(* CODESYS project BATW_Base0.0.0.33.library
   Company: Beckhoff Automation
   DefaultNamespace: BATW_Base
   Version: 0.0.0.33
   Placeholder: BATW_Base
   Author: BATW
   Description: Base library of BATW use
   Title: BATW_Base

Project tree, tasks and I/O mapping:
  libraries: Common Behaviour Model, * (3S - Smart Software Solutions GmbH); Tc2_Standard, * (Beckhoff Automation GmbH); Tc2_System, * (Beckhoff Automation GmbH); Tc2_Utilities, * (Beckhoff Automation GmbH); Tc3_EventLogger, * (Beckhoff Automation GmbH); Tc3_JsonXml, * (Beckhoff Automation GmbH); Tc3_Module, * (Beckhoff Automation GmbH)
  CBML_BASE/
    Behaviour-Model_Enums_STATE.png
    function block FB_ActionBasic [ST]: ControlCleanupAction, ControlCyclicAction, ControlExitAction, ControlResetAction, ControlStartAction, CleanupAction, CyclicAction, ExitAction, ResetAction, StartAction, IBehaviourModel, Get_ModelState, GetName
    function block FB_ActionBasic_Logger [ST]: M_ClearAlarm, M_ConfirmAlarm, M_ConnectAlarmLogger, M_RaiseAlarm, M_SetAlarmEvent, pAlarmState, M_AddEventMsg, M_ConnectMsgLogger, M_SetMessageEvent, M_AddJsonMsg, M_ConnectJsonMsgLogger
    interface I_BaseElement: Get_ModelState, GetName, IBehaviourModel
  00000000-0000-0000-0000-000000000000|CBML_BASE\Behaviour-Model_Enums_STATE.png
  Componets/
    DUTs/
      data type E_CylinderType
      data type ST_CylinderPara
    DUTs_Motor/
      data type ST_MotorPara
    function block FB_Cylinder [ST]: CleanupAction, CyclicAction, ExitAction, ResetAction, StartAction, EnableSimulation, IsDoubleValve, M_Extend, M_GetErrorMsg, M_Reset, M_Retract
    function block FB_Motor [ST]: CleanupAction, CyclicAction, ExitAction, ResetAction, StartAction, M_MotorStop, M_MoveBackward, M_MoveForward, M_Reset
  EventLogger/
    _Interface/
      Exporter/
        interface ITF_EventLogger_Exporter: M_ExportCSV
        interface ITF_EventLogger_Exporter_Carrier: M_ConnectExporter
      Logger/
        interface ITF_EventLogger_Alarm: M_ClearAlarm, M_ConfirmAlarm, M_RaiseAlarm, M_SetAlarmEvent, pAlarmState
        interface ITF_EventLogger_Alarm_Carrier: M_ClearAlarm, M_ConfirmAlarm, M_ConnectAlarmLogger, M_RaiseAlarm, M_SetAlarmEvent, pAlarmState
        interface ITF_EventLogger_Message: M_AddEventMsg, M_SetMessageEvent
        interface ITF_EventLogger_Message_Carrier: M_AddEventMsg, M_ConnectMsgLogger, M_SetMessageEvent
    _Test/
      program Demo_EventLogger [ST]
      function block FB_LoggerTest [ST]
    DUTs/
      data type E_EventExportType
      data type E_EventLanguage
      data type ST_AlarmEvent_State
    global variables EventLogger_Parameter
    function block FB_EventLogger_Alarm [ST]: M_ClearAlarm, M_ConfirmAlarm, M_RaiseAlarm, M_SetAlarmEvent, pAlarmState
    function block FB_EventLogger_Exporter [ST]: CleanupAction, CyclicAction, StartAction, M_SetCSV, M_SetExportLanguage, M_SetExportParameter
    function block FB_EventLogger_Message [ST]: M_AddEventMsg, M_SetMessageEvent
    program PRG_EventLogger [ST]: M_ExportLoggedEvent_Off, M_ExportLoggedEvent_On, M_ExportLoggedEvent_State, M_AlarmEvent_Init, M_MessageEvent_Init
  IO-Module/
    EL1889/
      data type ST_EL1889
      data type ST_EL1889_InfoData
      data type ST_EL1889_WcState
    EL2889/
      data type ST_EL2889
  JsonMsgLogger/
    _Interface/
      Client/
        interface ITF_AddJsonMsg_Behavior: M_AddJsonMsg
        interface ITF_GetJsonMsg_Behavior: M_GetJsonMsg
        interface ITF_JsonMSg_Carrier: M_ConnectJsonMsgLogger
        interface ITF_JsonMsg_Logger: M_AddJsonMsg, M_GetJsonMsg, pQueueAmount
      Server/
        interface ITF_JsonMsg_Handler: M_AttachJsonMsgLogger
    _Test/
      program Demo_JsonMsg [ST]
      function block FB_UserUnit [ST]
    Basic_Json/
      function block FB_Json_Converter [ST]: JsonStrToObj, ObjToJsonStr
      data type ST_Json_MsgLogger
    Basic_Queue/
      function block FB_Queue [ST]: dequeueElement, enqueueElement, enqueueElementfromHead, readElementbyIndex, readNextElement, releaseQueue, changeCurrentbyIndex, checkInputErr, deleteElement, moveCurrent2Next, moveCurrent2Prev, bIsQueueCreated, getDataTypebyIndex, getNextDataType, pGetHead, pGetTail, udiGetQueuedAmount
      data type ST_Queue
    data type E_HandlerQueueType
    data type E_LoggerQueueType
    data type E_OS_Type
    function block FB_JsonMsg_Handler [ST]: CleanupAction, CyclicAction, StartAction, M_AddJsonMsg, M_GetFilePathByTime, M_HandleMessage, FB_init, M_AttachJsonMsgLogger, M_SetFilePath
    function block FB_JsonMsg_Logger [ST]: M_AddJsonMsg, M_GetJsonMsg, pQueueAmount
    global variables JsonMsg_Parameter
    program PRG_JsonMsg [ST]: M_JsonMsg_Init, M_JsonMsg_SetFilePath
  POUs/
    program Demo [ST]
  Utilities/
    function block FB_EdgeDetect [ST]
  VISUs/
*)

// Componets/DUTs/E_CylinderType
{attribute 'qualified_only'}
{attribute 'strict'}
TYPE
    E_CylinderType :
    (
        Undefined    := 0,
        NoSensor     := 1,
        FrontSensor  := 2,
        RearSensor   := 3,
        DoubleSensor := 4
        );
END_TYPE

// Componets/DUTs/ST_CylinderPara
TYPE
    ST_CylinderPara :
    STRUCT
        ExtendTime       : TIME := T#0.2S;
        RetractTime      : TIME := T#0.2S;
        ExtendDelayTime  : TIME := T#0S;
        RetractDelayTime : TIME := T#0S;
        ExtendOverTime   : TIME := T#5S;
        RetractOverTime  : TIME := T#5S;
    END_STRUCT
END_TYPE

// Componets/DUTs_Motor/ST_MotorPara
TYPE ST_MotorPara :
STRUCT
	AccelerationTime : TIME := T#0.2S;
	DecelerationTime : TIME := T#0.4S;
END_STRUCT
END_TYPE

// EventLogger/DUTs/E_EventExportType
{attribute 'qualified_only'}
{attribute 'strict'}
TYPE E_EventExportType :
(
	Message_And_Alarm := 0,
	Message := 1,
	Alarm := 2
);
END_TYPE

// EventLogger/DUTs/E_EventLanguage
{attribute 'qualified_only'}
{attribute 'strict'}
TYPE E_EventLanguage :
(
	Chinese		:=1028,
	German		:=1031,
	English		:=1033
);
END_TYPE

// EventLogger/DUTs/ST_AlarmEvent_State
TYPE ST_AlarmEvent_State :
STRUCT
	bActive			: BOOL;
	bRaised			: BOOL;
	eConfirmnState	: TcEventConfirmationState;
	nTimeCleared	: ULINT;
	nTimeConfirm	: ULINT;
	nTimeRaised		: ULINT;
END_STRUCT
END_TYPE

// IO-Module/EL1889/ST_EL1889
TYPE ST_EL1889 :
STRUCT
        DI1  AT %I* :BIT;
        DI2  AT %I* :BIT;
        DI3  AT %I* :BIT;
        DI4  AT %I* :BIT;
        DI5  AT %I* :BIT;
        DI6  AT %I* :BIT;
        DI7  AT %I* :BIT;
        DI8  AT %I* :BIT;
        DI9  AT %I* :BIT;
        DI10 AT %I* :BIT;
        DI11 AT %I* :BIT;
        DI12 AT %I* :BIT;
        DI13 AT %I* :BIT;
        DI14 AT %I* :BIT;
        DI15 AT %I* :BIT;
        DI16 AT %I* :BIT;
		WcState AT%I*:ST_EL1889_WcState;
		InfoData AT%I*:UINT;
END_STRUCT
END_TYPE

// IO-Module/EL1889/ST_EL1889_InfoData
TYPE ST_EL1889_InfoData :
STRUCT
	
END_STRUCT
END_TYPE

// IO-Module/EL1889/ST_EL1889_WcState
TYPE ST_EL1889_WcState :
STRUCT
	WcState : BIT;
	InputToggle:BIT;
END_STRUCT
END_TYPE

// IO-Module/EL2889/ST_EL2889
TYPE ST_EL2889 :
STRUCT
	WcState AT%Q*: BIT;
	
END_STRUCT
END_TYPE

// JsonMsgLogger/Basic_Json/ST_Json_MsgLogger
TYPE ST_Json_MsgLogger :
STRUCT
	tTime		:STRING;//DT;
	{attribute 'TcEncoding':='UTF-8'}
	sMessage	:T_MaxString;
END_STRUCT
END_TYPE

// JsonMsgLogger/Basic_Queue/ST_Queue
{attribute 'enable_dynamic_creation'}
{attribute 'pack_mode' := '0'}
TYPE ST_Queue :
STRUCT
	iDataType:INT;
	pData  :POINTER TO BYTE; //Current data addr
	pPrev  :POINTER TO ST_Queue; //Previous addr
	pNext  :POINTER TO ST_Queue; //Next addr
END_STRUCT
END_TYPE

// JsonMsgLogger/E_HandlerQueueType
{attribute 'qualified_only'}
{attribute 'strict'}
TYPE E_HandlerQueueType :
(
	RingBuffer 		:=0,
	Queue			:=1
);
END_TYPE

// JsonMsgLogger/E_LoggerQueueType
{attribute 'qualified_only'}
{attribute 'strict'}
TYPE E_LoggerQueueType :
(
	RingBuffer 		:=0,
	FixedSizeArray	:=1,
	Queue			:=2
);
END_TYPE

// JsonMsgLogger/E_OS_Type
{attribute 'qualified_only'}
{attribute 'strict'}
TYPE E_OS_Type :
(
	WinCE :=0,
	Windows:=1
);
END_TYPE

// EventLogger/EventLogger_Parameter
VAR_GLOBAL CONSTANT
	uiAlarmEventNum				:UINT:=200;//Machine Alarm Event Num
	uiMessageEventNum			:UINT:=1;//Machine Message Event Num
END_VAR

// JsonMsgLogger/JsonMsg_Parameter
//{attribute 'qualified_only'}
VAR_GLOBAL CONSTANT
	
	(* System *)
	eOsType							:E_OS_Type:=E_OS_Type.Windows;
	
	(* Logger/Handler *)
	uiHandlerNum					:UINT:=5;
	uiLoggerNum						:UINT:=200;
	uiLoggerInHandlerMaxNum			:UINT:=200;
	
	
	(*Multiply 2 var below, is the MAX Message Handle num Per Cycle*)
	uiLoggerHandleLimitPerCycle		:UINT:=10;//One Cycle can deal with N Logger's all queued msg
	uiMsgHandleLimitPerLogger		:UINT:=200;//when exceed this value, pass to next subject,prevent from starving
	
	
	(* Logger BufferSize *)
	eLoggerQueueType	:E_LoggerQueueType := E_LoggerQueueType.RingBuffer;
	uiBufferSize		:UINT:=1000;
	uiRingBufferSize	:UINT:=10*1000;//10 K Bytes
	
	
	(* Handler BufferSize *)
	eHandlerQueueType		:E_HandlerQueueType := E_HandlerQueueType.RingBuffer;
	uiHandlerRingBufferSize	:UDINT:=3*1000*1000;//3M Bytes
	
	
END_VAR

// CBML_BASE/FB_ActionBasic
{attribute 'reflection'}
FUNCTION_BLOCK FB_ActionBasic IMPLEMENTS I_BaseElement, CBML.IActionController,CBML.IActionProvider
VAR_INPUT
END_VAR
VAR_OUTPUT
    xDone  : BOOL; // True: Ready condition reached
    xBusy  : BOOL; // True: Operation is running
    xError : BOOL; // True: Error condition reached
END_VAR
VAR
    {attribute 'instance-path'} 
    {attribute 'noinit'}
    _strName: STRING(255); 					// Instance path of the FB for Diagnostic
	
	_ActionController : CBML.ActionController;
	_iBehaviourModel : CBML.IBehaviourModel;
END_VAR

(* An action controller is used whenever it is necessary to have the actions of the action controller
 instead of those of the action provider called. ``ControlCleanupAction`` is the action controller
 specifically used to control the |STATE.CLEANING| state.*)
METHOD ControlCleanupAction
VAR_INPUT
	itfCleanupActionProvider	: CBML.ICleanupActionProvider;
	xAbortProposed	: BOOL;
	iErrorIDProposed	: INT;
END_VAR
VAR_OUTPUT
	xComplete	: BOOL;
	xAbort	: BOOL;
	iErrorID	: INT;
END_VAR
CleanupAction(xAbortProposed:= xAbortProposed, iErrorIDProposed:= iErrorIDProposed, xComplete=> xComplete, xAbort=> xAbort, iErrorID=> iErrorID);
END_METHOD

(* An action controller is used whenever it is necessary to have the actions of the action controller
 instead of those of the action provider called. ``ControlCyclicAction`` is the action controller
 specifically used to control the |STATE.EXECUTING| state.*)
METHOD ControlCyclicAction
VAR_INPUT
	itfCyclicActionProvider	: CBML.ICyclicActionProvider;
	itfTimingController	: CBML.ITimingController;
END_VAR
VAR_OUTPUT
	xComplete	: BOOL;
	iErrorID	: INT;
END_VAR
CyclicAction(itfTimingController:= itfTimingController, xComplete=> xComplete, iErrorID=> iErrorID);
END_METHOD

(* Intended for releasing external resources (like RTS handles)

 Do not call other internal function block instances in the context of this method.
 Call only external functions defined inside the RTS.
 For cleaning up other resources than external ones, please use the ``CleanupAction``.
 This method should be callable in the context of ``FB_EXIT`` for example
 before downloading a new application or before reseting an application.*)
METHOD ControlExitAction
VAR_INPUT
	itfExitActionProvider	: CBML.IExitActionProvider;
	xAfterCleanup	: BOOL;
	xInCopyCode	: BOOL;
END_VAR
ExitAction(xAfterCleanup:= xAfterCleanup, xInCopyCode:= xInCopyCode);
END_METHOD

(* An action controller is used whenever it is necessary to have the actions of the action controller
 instead of those of the action provider called. ``ControlResetAction`` is the action controller
 specifically used to control the |STATE.RESETTING| state.*)
METHOD ControlResetAction
VAR_INPUT
	itfResetActionProvider	: CBML.IResetActionProvider;
END_VAR
VAR_OUTPUT
	xComplete	: BOOL;
END_VAR
ResetAction(xComplete=> xComplete);
END_METHOD

(* An action controller is used whenever it is necessary to have the actions of the action controller
 instead of those of the action provider called. ``ControlStartAction`` is the action controller
 specifically used to control the |STATE.STARTING| state.*)
METHOD ControlStartAction
VAR_INPUT
	itfStartActionProvider	: CBML.IStartActionProvider;
END_VAR
VAR_OUTPUT
	xComplete	: BOOL;
	iErrorID	: INT;
END_VAR
StartAction(xComplete=> xComplete, iErrorID=> iErrorID);
END_METHOD

METHOD CleanupAction
VAR_INPUT
    xAbortProposed : BOOL;
    iErrorIDProposed: INT;
END_VAR
VAR_OUTPUT
    xComplete : BOOL := TRUE;
    xAbort: BOOL := xAbortProposed;
 	iErrorID : INT := iErrorIDProposed;
END_VAR
END_METHOD

METHOD CyclicAction
VAR_INPUT
    itfTimingController : CBML.ITimingController;
END_VAR
VAR_OUTPUT
    xComplete : BOOL := TRUE;
    iErrorID : INT := 0;
END_VAR
END_METHOD

METHOD ExitAction
VAR_INPUT
    xAfterCleanup : BOOL;
    xInCopyCode : BOOL;
END_VAR
END_METHOD

METHOD ResetAction
VAR_OUTPUT
    xComplete : BOOL := TRUE;
END_VAR
END_METHOD

METHOD StartAction
VAR_OUTPUT
    xComplete : BOOL := TRUE;
	iErrorID : INT := 0;
END_VAR
END_METHOD

PROPERTY IBehaviourModel : CBML.IBehaviourModel
GET
IBehaviourModel:= _iBehaviourModel;
END_GET
SET
_iBehaviourModel := IBehaviourModel;
IBehaviourModel.ActionController := THIS^;
END_SET
END_PROPERTY

METHOD Get_ModelState
VAR_INPUT
    xCommit : BOOL;
END_VAR
VAR_OUTPUT
    xDone : BOOL;
    xBusy : BOOL;
    xError : BOOL;
    xAborted : BOOL;
    iErrorID : INT;
    eState : CBML.STATE;
END_VAR
END_METHOD

METHOD GetName : STRING
VAR_INPUT
END_VAR
END_METHOD

END_FUNCTION_BLOCK

// CBML_BASE/I_BaseElement
INTERFACE I_BaseElement EXTENDS __SYSTEM.IQueryInterface

METHOD Get_ModelState
VAR_INPUT
    xCommit : BOOL;
END_VAR
VAR_OUTPUT
    xDone : BOOL;
    xBusy : BOOL;
    xError : BOOL;
    xAborted : BOOL;
    iErrorID : INT;
    eState : CBML.STATE;
END_VAR
END_METHOD

METHOD GetName : STRING
VAR_INPUT
END_VAR
END_METHOD

PROPERTY IBehaviourModel : CBML.IBehaviourModel
GET
END_GET
SET
END_SET
END_PROPERTY

END_INTERFACE

// CBML_BASE/FB_ActionBasic_Logger
FUNCTION_BLOCK FB_ActionBasic_Logger EXTENDS FB_ActionBasic
IMPLEMENTS 
	(*Json Msg *)
	ITF_JsonMSg_Carrier,ITF_AddJsonMsg_Behavior,
	(* EventLogger *)
	ITF_EventLogger_Alarm_Carrier,ITF_EventLogger_Message_Carrier
VAR_INPUT
END_VAR
VAR_OUTPUT
END_VAR
VAR
	(*-----Json Message-----*)
	itfJsonMsgLogger			:ITF_JsonMsg_Logger;
	
	(*-----EventLogger-----*)
	itfEventLogger_Alarm		:ITF_EventLogger_Alarm;(* Alarm *)
	itfEventLogger_Message		:ITF_EventLogger_Message;(* Message *)
END_VAR

METHOD M_ClearAlarm : BOOL
VAR_OUTPUT
	iErrorID	: INT;
END_VAR
IF itfEventLogger_Alarm <> 0 THEN
	itfEventLogger_Alarm.M_ClearAlarm(iErrorID => iErrorID);
ELSE
	iErrorID:=9999;
END_IF
END_METHOD

METHOD M_ConfirmAlarm : BOOL
VAR_OUTPUT
	iErrorID	: INT;
END_VAR
IF itfEventLogger_Alarm <> 0 THEN
	itfEventLogger_Alarm.M_ConfirmAlarm(iErrorID => iErrorID);
ELSE
	iErrorID:=9999;
END_IF
END_METHOD

METHOD M_ConnectAlarmLogger : BOOL
VAR_INPUT
	IDevice	: ITF_EventLogger_Alarm;
END_VAR
VAR_OUTPUT
	iErrorID : INT := 0;
END_VAR
IF IDevice <> 0 THEN
	THIS^.itfEventLogger_Alarm := IDevice;
ELSE
	iErrorID := 9999;
END_IF
END_METHOD

METHOD M_RaiseAlarm : BOOL
VAR_INPUT
	sLogMessage	: T_MaxString;
END_VAR
VAR_OUTPUT
	iErrorID	: INT;
END_VAR
IF itfEventLogger_Alarm <> 0 THEN
	itfEventLogger_Alarm.M_RaiseAlarm(THIS^._strName, 0, sLogMessage, iErrorID => iErrorID);
ELSE
	iErrorID:=9999;
END_IF
END_METHOD

METHOD M_SetAlarmEvent : BOOL
VAR_INPUT
	Event	: TcEventEntry;
END_VAR
VAR_OUTPUT
    iErrorID : INT;
END_VAR
IF itfEventLogger_Alarm <> 0 THEN
	itfEventLogger_Alarm.M_SetAlarmEvent(Event, iErrorID => iErrorID);
ELSE
	iErrorID:=9999;
END_IF
END_METHOD

PROPERTY pAlarmState : ST_AlarmEvent_State
GET
pAlarmState := THIS^.itfEventLogger_Alarm.pAlarmState;
END_GET
END_PROPERTY

METHOD M_AddEventMsg : BOOL
VAR_INPUT
	sLogMessage	:T_MaxString;
END_VAR
VAR_OUTPUT
	iErrorID : INT := 0;
END_VAR
IF itfEventLogger_Message <> 0 THEN
	itfEventLogger_Message.M_AddEventMsg(THIS^._strName, 0, sLogMessage, iErrorID => iErrorID);
ELSE
	iErrorID:=9999;
END_IF
END_METHOD

METHOD M_ConnectMsgLogger : BOOL
VAR_INPUT
	IDevice	:ITF_EventLogger_Message;
END_VAR
VAR_OUTPUT
	iErrorID : INT := 0;
END_VAR
IF IDevice <> 0 THEN
	THIS^.itfEventLogger_Message := IDevice;
	M_ConnectMsgLogger:=TRUE;
ELSE
	M_ConnectMsgLogger:=FALSE;
END_IF
END_METHOD

METHOD M_SetMessageEvent : BOOL
VAR_INPUT
	Event	: TcEventEntry;
END_VAR
VAR_OUTPUT
	iErrorID	: INT;
END_VAR
IF itfEventLogger_Message <> 0 THEN
	itfEventLogger_Message.M_SetMessageEvent(Event, iErrorID => iErrorID);
ELSE
	iErrorID:=9999;
END_IF
END_METHOD

METHOD M_AddJsonMsg : BOOL
VAR_INPUT
	sLogMsg	: T_MaxString;
END_VAR
VAR_OUTPUT
	uiResult	: UINT;
END_VAR
itfJsonMsgLogger.M_AddJsonMsg(sLogMsg := sLogMsg, uiResult => uiResult);
END_METHOD

METHOD M_ConnectJsonMsgLogger : BOOL
VAR_INPUT
	IDevice	: ITF_JsonMsg_Logger;
END_VAR
IF IDevice <> 0 THEN
	THIS^.itfJsonMsgLogger := IDevice;
	M_ConnectJsonMsgLogger:=TRUE;
ELSE
	M_ConnectJsonMsgLogger:=FALSE;
END_IF
END_METHOD

END_FUNCTION_BLOCK

// JsonMsgLogger/_Interface/Client/ITF_JsonMSg_Carrier
INTERFACE ITF_JsonMSg_Carrier

METHOD M_ConnectJsonMsgLogger : BOOL
VAR_INPUT
	IDevice	:ITF_JsonMsg_Logger;
END_VAR
END_METHOD

END_INTERFACE

// JsonMsgLogger/_Interface/Client/ITF_JsonMsg_Logger
INTERFACE ITF_JsonMsg_Logger

METHOD M_AddJsonMsg : BOOL
VAR_INPUT
	sLogMsg			:T_MaxString;
END_VAR
VAR_OUTPUT
	uiResult:UINT;
END_VAR
END_METHOD

METHOD M_GetJsonMsg : BOOL
VAR_OUTPUT
	stJsonMsg	:ST_Json_MsgLogger;
	uiResult	:UINT;
END_VAR
END_METHOD

PROPERTY pQueueAmount : uint
GET
END_GET
END_PROPERTY

END_INTERFACE

// JsonMsgLogger/_Interface/Client/ITF_AddJsonMsg_Behavior
INTERFACE ITF_AddJsonMsg_Behavior

METHOD M_AddJsonMsg : BOOL
VAR_INPUT
	sLogMsg			:T_MaxString;
END_VAR
VAR_OUTPUT
	uiResult:UINT;
END_VAR
END_METHOD

END_INTERFACE

// EventLogger/_Interface/Logger/ITF_EventLogger_Alarm_Carrier
INTERFACE ITF_EventLogger_Alarm_Carrier

METHOD M_ClearAlarm : BOOL
VAR_INPUT
END_VAR
VAR_OUTPUT
    iErrorID : INT;
END_VAR
END_METHOD

METHOD M_ConfirmAlarm : BOOL
VAR_INPUT
END_VAR
VAR_OUTPUT
    iErrorID : INT;
END_VAR
END_METHOD

METHOD M_ConnectAlarmLogger : BOOL
VAR_INPUT
	IDevice	:ITF_EventLogger_Alarm;
END_VAR
VAR_OUTPUT
	iErrorID : INT;
END_VAR
END_METHOD

METHOD M_RaiseAlarm : BOOL
VAR_INPUT
	sLogMessage		: T_MaxString;
END_VAR
VAR_OUTPUT
    iErrorID : INT;
END_VAR
END_METHOD

METHOD M_SetAlarmEvent : BOOL
VAR_INPUT
	Event	:TcEventEntry;
END_VAR
VAR_OUTPUT
    iErrorID : INT;
END_VAR
END_METHOD

PROPERTY pAlarmState : ST_AlarmEvent_State
GET
END_GET
END_PROPERTY

END_INTERFACE

// EventLogger/_Interface/Logger/ITF_EventLogger_Alarm
INTERFACE ITF_EventLogger_Alarm

METHOD M_ClearAlarm : BOOL
VAR_INPUT
END_VAR
VAR_OUTPUT
    iErrorID : INT;
END_VAR
END_METHOD

METHOD M_ConfirmAlarm : BOOL
VAR_INPUT
END_VAR
VAR_OUTPUT
    iErrorID : INT;
END_VAR
END_METHOD

METHOD M_RaiseAlarm : BOOL
VAR_INPUT
	sSource_Name	: STRING(255);
	nSource_Id		: UDINT;
	sLogMessage		: T_MaxString;
END_VAR
VAR_OUTPUT
    iErrorID : INT;
END_VAR
END_METHOD

METHOD M_SetAlarmEvent : BOOL
VAR_INPUT
	Event	:TcEventEntry;
END_VAR
VAR_OUTPUT
    iErrorID : INT;
END_VAR
END_METHOD

PROPERTY pAlarmState : ST_AlarmEvent_State
GET
END_GET
END_PROPERTY

END_INTERFACE

// EventLogger/_Interface/Logger/ITF_EventLogger_Message_Carrier
INTERFACE ITF_EventLogger_Message_Carrier

METHOD M_AddEventMsg : BOOL
VAR_INPUT
	sLogMessage	:T_MaxString;
END_VAR
VAR_OUTPUT
	iErrorID : INT;
END_VAR
END_METHOD

METHOD M_ConnectMsgLogger : BOOL
VAR_INPUT
	IDevice	:ITF_EventLogger_Message;
END_VAR
VAR_OUTPUT
	iErrorID : INT;
END_VAR
END_METHOD

METHOD M_SetMessageEvent : BOOL
VAR_INPUT
	Event	:TcEventEntry;
END_VAR
VAR_OUTPUT
    iErrorID : INT;
END_VAR
END_METHOD

END_INTERFACE

// EventLogger/_Interface/Logger/ITF_EventLogger_Message
INTERFACE ITF_EventLogger_Message

METHOD M_AddEventMsg : BOOL
VAR_INPUT
	//Event			:TcEventEntry;
	sSource_Name	:STRING(255);
	nSource_Id		:UDINT;
	sLogMessage		:T_MaxString;
END_VAR
VAR_OUTPUT
	iErrorID : INT;
END_VAR
END_METHOD

METHOD M_SetMessageEvent : BOOL
VAR_INPUT
	Event	:TcEventEntry;
END_VAR
VAR_OUTPUT
    iErrorID : INT;
END_VAR
END_METHOD

END_INTERFACE

// Componets/FB_Cylinder
{attribute 'reflection'}
FUNCTION_BLOCK FB_Cylinder EXTENDS FB_ActionBasic
VAR_INPUT
    xEnable     : BOOL; // True : Active this cylinder component service
    FrontSensor : BOOL; // Input position for the Front Sensor, used to read external signals. 
    RearSensor  : BOOL; // Input position for the Rear Sensor, used to read external signals.
    SetupPara   : ST_CylinderPara;
END_VAR
VAR_OUTPUT
    CurrentCylinderType : E_CylinderType;
    InFrontPosition     : BOOL; // 到達前極限
    InRearPosition      : BOOL;
    ExtendOutput        : BOOL;
    RetractOutput       : BOOL;
    iErrorID            : INT;
    ErrorMsg              : STRING;
END_VAR
VAR
    // State Machine
    StateBehaviour : CBML.LConC;
    // Sensor Check
    {attribute 'is_connected' := 'FrontSensor'}
    FrontSensor_IsConnected : BOOL;
    {attribute 'is_connected' := 'RearSensor'}
    RearSensor_IsConnected : BOOL;

    // internal
    ExtendCMD      : BOOL;
    _IsDoubleValve : BOOL;
    _IsSimulation  : BOOL;
    // Timer 
    TON_Extend            : TON;
    TON_Retracted         : TON;
    TON_ExtendDelay       : TON;
    TON_RetractedDelay    : TON;
    TON_ExtendOverTime    : TON;
    TON_RetractedOverTime : TON;
END_VAR

THIS^.IBehaviourModel := StateBehaviour;
StateBehaviour(xEnable := xEnable, xBusy => xBusy, xError => xError);

TON_Extend(PT := SetupPara.ExtendTime);
TON_Retracted(PT := SetupPara.RetractTime);
TON_ExtendDelay(PT := SetupPara.ExtendDelayTime);
TON_RetractedDelay(PT := SetupPara.RetractDelayTime);
TON_ExtendOverTime(PT := SetupPara.ExtendOverTime);
TON_RetractedOverTime(PT := SetupPara.RetractOverTime);

iErrorID := StateBehaviour._model.iErrorID;
ErrorMsg := M_GetErrorMsg(xErrorID := iErrorID);

METHOD PRIVATE CleanupAction
VAR_INPUT
    xAbortProposed : BOOL;
    iErrorIDProposed: INT;
	
END_VAR
VAR_OUTPUT
    xComplete : BOOL := TRUE;
    xAbort: BOOL := xAbortProposed;
 	iErrorID : INT := iErrorIDProposed;
END_VAR
(* This action is used to release all resource
*)
ExtendOutput := FALSE;
RetractOutput := FALSE;
Ton_Extend.IN            := FALSE;
TON_Retracted.IN         := FALSE;
TON_ExtendDelay.IN       := FALSE;
TON_RetractedDelay.IN    := FALSE;
TON_ExtendOverTime.IN    := FALSE;
TON_RetractedOverTime.IN := FALSE;
END_METHOD

METHOD PRIVATE CyclicAction
VAR_INPUT
    itfTimingController : CBML.ITimingController;
END_VAR
VAR_OUTPUT
    xComplete : BOOL := TRUE;
    iErrorID : INT := 0;
END_VAR
IF ExtendCMD THEN
    IF NOT _IsDoubleValve THEN
        ExtendOutput := TRUE;
        RetractOutput := FALSE;
    ELSE
        ExtendOutput := NOT InFrontPosition;
        RetractOutput := FALSE;
    END_IF
ELSE
    IF NOT _IsDoubleValve THEN
        ExtendOutput := FALSE;
        RetractOutput := TRUE;
    ELSE
        ExtendOutput := FALSE;
        RetractOutput := NOT InRearPosition;
    END_IF
END_IF

(* Valve control *)
Ton_Extend.IN := ExtendOutput;
TON_Retracted.IN := RetractOutput;
TON_ExtendDelay.IN := (FrontSensor_IsConnected AND (FrontSensor)) OR ((NOT FrontSensor_IsConnected OR _IsSimulation) AND Ton_Extend.Q);
TON_RetractedDelay.IN := (RearSensor_IsConnected AND (RearSensor)) OR ((NOT RearSensor_IsConnected OR _IsSimulation) AND TON_Retracted.Q);
TON_ExtendOverTime.IN := ExtendOutput AND NOT TON_ExtendDelay.Q;
TON_RetractedOverTime.IN := RetractOutput AND NOT TON_RetractedDelay.Q;

CASE CurrentCylinderType OF
    E_CylinderType.NoSensor:
		IF TON_ExtendDelay.Q THEN
			InFrontPosition := TRUE;
		ELSIF RetractOutput THEN
			InFrontPosition := FALSE;
		END_IF
		IF TON_RetractedDelay.Q THEN
			InRearPosition := TRUE;
		ELSIF ExtendOutput THEN
			InRearPosition := FALSE;
		END_IF
    E_CylinderType.FrontSensor:
        InFrontPosition := FrontSensor;
		
		IF TON_RetractedDelay.Q THEN
			InRearPosition := TRUE;
		ELSIF ExtendOutput THEN
			InRearPosition := FALSE;
		END_IF
    E_CylinderType.RearSensor:
		IF TON_ExtendDelay.Q THEN
			InFrontPosition := TRUE;
		ELSIF RetractOutput THEN
			InFrontPosition := FALSE;
		END_IF
        InRearPosition := RearSensor;
    E_CylinderType.DoubleSensor:
        InFrontPosition := FrontSensor;
        InRearPosition := RearSensor;
END_CASE

(* Error handler *)
IF TON_ExtendOverTime.Q THEN
    iErrorID := 2; // Extend time out
ELSIF TON_RetractedOverTime.Q THEN
    iErrorID := 3; // Retract time out
ELSE
    iErrorID := 0; // No Error
END_IF
END_METHOD

METHOD PRIVATE ExitAction
VAR_INPUT
    xAfterCleanup : BOOL;
    xInCopyCode : BOOL;
END_VAR
END_METHOD

METHOD PRIVATE ResetAction
VAR_OUTPUT
    xComplete : BOOL := TRUE;
END_VAR
InFrontPosition := FALSE;
InRearPosition  := FALSE;
END_METHOD

METHOD PRIVATE StartAction
VAR_OUTPUT
    xComplete : BOOL := TRUE;
	iErrorID : INT := 0;
END_VAR
IF NOT _IsSimulation THEN
    IF NOT FrontSensor_IsConnected AND NOT RearSensor_IsConnected THEN
        CurrentCylinderType := E_CylinderType.NoSensor;
        iErrorID := 0;
    ELSIF FrontSensor_IsConnected AND NOT RearSensor_IsConnected THEN
        CurrentCylinderType := E_CylinderType.FrontSensor;
        iErrorID := 0;
    ELSIF NOT FrontSensor_IsConnected AND RearSensor_IsConnected THEN
        CurrentCylinderType := E_CylinderType.RearSensor;
        iErrorID := 0;
    ELSIF FrontSensor_IsConnected AND RearSensor_IsConnected THEN
        CurrentCylinderType := E_CylinderType.DoubleSensor;
        iErrorID := 0;
    END_IF
ELSE
    CurrentCylinderType := E_CylinderType.NoSensor;
    iErrorID := 0;
END_IF
END_METHOD

PROPERTY EnableSimulation : Bool
SET
_IsSimulation := EnableSimulation ;
END_SET
END_PROPERTY

PROPERTY IsDoubleValve : bool
SET
_IsDoubleValve := IsDoubleValve;
END_SET
END_PROPERTY

METHOD PUBLIC M_Extend
VAR_INPUT
END_VAR
ExtendCMD := TRUE;
END_METHOD

METHOD M_GetErrorMsg : T_MaxString
VAR_INPUT
	xErrorID: INT;
END_VAR

VAR
	
END_VAR
CASE xErrorID OF
    0:
        M_GetErrorMsg := 'No Error';
    1:
        M_GetErrorMsg := 'Action time out';
    2:
        M_GetErrorMsg := 'Extend time out';
	3:
		M_GetErrorMsg := 'Retract time out';
END_CASE
END_METHOD

METHOD PUBLIC M_Reset
VAR_INPUT
END_VAR
VAR
	ExecuteReset :BOOL := true;
END_VAR
StateBehaviour.ResetModel(xCommit:=ExecuteReset);
END_METHOD

METHOD PUBLIC M_Retract
VAR_INPUT
END_VAR
ExtendCMD := FALSE;
END_METHOD

END_FUNCTION_BLOCK

// Componets/FB_Motor
FUNCTION_BLOCK FB_Motor EXTENDS FB_ActionBasic
VAR_INPUT
    xEnable          : BOOL; // True : Active this cylinder component service
	OverLoadSignal : BOOL;
	SetupPara : ST_MotorPara;
END_VAR
VAR_OUTPUT
	InForWard :BOOL;
	InBackWard : BOOL;
	InStopped :BOOL;
	ForWardOutput : BOOL;
	BackWardOutput : BOOL;
END_VAR
VAR
    // State Machine
    StateBehaviour : CBML.LConC;

	{attribute 'is_connected' := 'OverLoadSignal'}
	OverLoadDetectActive : BOOL;
	// Timer
	TON_AccelerationTime : TON;
	TON_DecelerationTime : TON;
	ForwardCMD: BOOL;
	BackWardCMD: BOOL;
	
END_VAR

THIS^.IBehaviourModel := StateBehaviour;
StateBehaviour(xEnable := xEnable, xBusy => xBusy, xError => xError);

TON_AccelerationTime(IN:= , PT:= SetupPara.AccelerationTime, Q=> , ET=> );
TON_DecelerationTime(IN:= , PT:= SetupPara.DecelerationTime, Q=> , ET=> );

METHOD PRIVATE CleanupAction
VAR_INPUT
    xAbortProposed : BOOL;
    iErrorIDProposed: INT;
END_VAR
VAR_OUTPUT
    xComplete : BOOL := TRUE;
    xAbort: BOOL := xAbortProposed;
 	iErrorID : INT := iErrorIDProposed;
END_VAR
InForWard := FALSE;
InBackWard := FALSE;

ForWardOutput := FALSE;
BackWardOutput := FALSE;
TON_AccelerationTime.IN := FALSE;
TON_DecelerationTime.IN := FALSE;
END_METHOD

METHOD PRIVATE CyclicAction
VAR_INPUT
    itfTimingController : CBML.ITimingController;
END_VAR
VAR_OUTPUT
    xComplete : BOOL := TRUE;
    iErrorID : INT := 0;
END_VAR
IF ForwardCMD AND NOT BackWardCMD THEN
    ForWardOutput := TRUE;
    BackWardOutput := FALSE;
ELSIF BackWardCMD AND NOT ForwardCMD THEN
    ForWardOutput := FALSE;
    BackWardOutput := TRUE;
ELSIF ForwardCMD AND BackWardCMD THEN
    ForWardOutput := FALSE;
    BackWardOutput := FALSE;
ELSE
    ForWardOutput := FALSE;
    BackWardOutput := FALSE;
END_IF

(* Output Control *)
TON_AccelerationTime.IN := ForWardOutput OR BackWardOutput;
TON_DecelerationTime.IN := NOT (ForWardOutput OR BackWardOutput);

InForWard := TON_AccelerationTime.Q AND ForWardOutput;
InBackWard := TON_AccelerationTime.Q AND BackWardOutput;
InStopped := TON_DecelerationTime.Q;
END_METHOD

METHOD PRIVATE ExitAction
VAR_INPUT
    xAfterCleanup : BOOL;
    xInCopyCode : BOOL;
END_VAR
END_METHOD

METHOD PRIVATE ResetAction
VAR_OUTPUT
    xComplete : BOOL := TRUE;
END_VAR
InForWard := FALSE;
InBackWard := FALSE;
END_METHOD

METHOD PRIVATE StartAction
VAR_OUTPUT
    xComplete : BOOL := TRUE;
	iErrorID : INT := 0;
END_VAR
END_METHOD

METHOD PUBLIC M_MotorStop
VAR_INPUT
END_VAR
ForwardCMD :=FALSE;
BackWardCMD := FALSE;
END_METHOD

METHOD PUBLIC M_MoveBackward
VAR_INPUT
END_VAR
ForwardCMD :=FALSE;
BackWardCMD := TRUE;
END_METHOD

METHOD PUBLIC M_MoveForward
VAR_INPUT
END_VAR
ForwardCMD :=TRUE;
BackWardCMD := FALSE;
END_METHOD

METHOD PUBLIC M_Reset
VAR_INPUT
END_VAR
VAR
    ExecuteReset : BOOL := TRUE;
END_VAR
StateBehaviour.ResetModel(xCommit:=ExecuteReset);
END_METHOD

END_FUNCTION_BLOCK

// EventLogger/_Interface/Exporter/ITF_EventLogger_Exporter
INTERFACE ITF_EventLogger_Exporter

METHOD M_ExportCSV : BOOL
VAR_INPUT
END_VAR
END_METHOD

END_INTERFACE

// EventLogger/_Interface/Exporter/ITF_EventLogger_Exporter_Carrier
INTERFACE ITF_EventLogger_Exporter_Carrier EXTENDS ITF_EventLogger_Exporter

METHOD M_ConnectExporter : BOOL
VAR_INPUT
END_VAR
END_METHOD

END_INTERFACE

// EventLogger/_Test/Demo_EventLogger
PROGRAM Demo_EventLogger
VAR
	fbTester	:ARRAY[0..10] OF FB_LoggerTest;
	fbTester222	:ARRAY[0..10] OF FB_LoggerTest;
	bTest		:BOOL;
	bExport		:BOOL;
	bDone		:BOOL;
END_VAR

(*----- 1. Program Call -----*)
PRG_EventLogger();

(*----- 2. Set Event and Connect to Device -----*)
(* Users need to build their own Event Classes in Type System before call these Init Functions. *)
PRG_EventLogger.M_MessageEvent_Init(fbTester[0], TC_EVENTS.MessageEvent_Demo.Message ,0);
PRG_EventLogger.M_MessageEvent_Init(fbTester[1], TC_EVENTS.MessageEvent_Demo.Message ,0);
PRG_EventLogger.M_MessageEvent_Init(fbTester[2], TC_EVENTS.MessageEvent_Demo.Message ,0);
PRG_EventLogger.M_MessageEvent_Init(fbTester[3], TC_EVENTS.MessageEvent_Demo.Message ,0);
PRG_EventLogger.M_MessageEvent_Init(fbTester222[0], TC_EVENTS.MessageEvent_Demo.Message ,0);
PRG_EventLogger.M_MessageEvent_Init(fbTester222[1], TC_EVENTS.MessageEvent_Demo.Message ,0);
PRG_EventLogger.M_MessageEvent_Init(fbTester222[2], TC_EVENTS.MessageEvent_Demo.Message ,0);
PRG_EventLogger.M_MessageEvent_Init(fbTester222[3], TC_EVENTS.MessageEvent_Demo.Message ,0);

PRG_EventLogger.M_AlarmEvent_Init(fbTester[0], TC_EVENTS.AlarmEvent_Demo.A0001_Alarm, 0);
PRG_EventLogger.M_AlarmEvent_Init(fbTester[1], TC_EVENTS.AlarmEvent_Demo.A0002_Alarm, 1);
PRG_EventLogger.M_AlarmEvent_Init(fbTester[2], TC_EVENTS.AlarmEvent_Demo.A0003_Alarm, 2);
PRG_EventLogger.M_AlarmEvent_Init(fbTester222[0], TC_EVENTS.AlarmEvent_Demo.A0004_Alarm, 3);
PRG_EventLogger.M_AlarmEvent_Init(fbTester222[1], TC_EVENTS.AlarmEvent_Demo.A0005_Alarm, 4);
PRG_EventLogger.M_AlarmEvent_Init(fbTester222[2], TC_EVENTS.AlarmEvent_Demo.A0006_Alarm, 5);
PRG_EventLogger.M_AlarmEvent_Init(fbTester222[3], TC_EVENTS.AlarmEvent_Demo.A0007_Alarm, 6);

(*----- 3. Demo Test -----*)
IF bTest THEN
	bTest:=FALSE;
	
	fbTester[2].M_AddEventMsg('Msg Before Alarm Raised');
	fbTester[2].M_RaiseAlarm('Alarm 123');
	fbTester222[3].M_AddEventMsg('Msg Before Alarm Raised');
	fbTester222[3].M_RaiseAlarm('Alarm 456');
END_IF

IF bExport THEN
	PRG_EventLogger.M_ExportLoggedEvent_On(E_EventExportType.Message_And_Alarm,'C:\Users\LeoL\Desktop\Test.CSV');
	
	PRG_EventLogger.M_ExportLoggedEvent_State(xDone => bDone);
	
	IF bDone THEN
		bExport:=false;
		PRG_EventLogger.M_ExportLoggedEvent_Off();
	END_IF
	
END_IF

END_PROGRAM

// EventLogger/PRG_EventLogger
PROGRAM PRG_EventLogger
VAR
	fbAlarmLogger			:ARRAY[0..uiAlarmEventNum-1] OF FB_EventLogger_Alarm;
	fbMessageLogger			:ARRAY[0..uiMessageEventNum-1] OF FB_EventLogger_Message;
	fbExporter				:FB_EventLogger_Exporter;
END_VAR
VAR
	i		:UINT;
END_VAR

fbExporter(xExecute:=);

FOR i:=0 TO uiAlarmEventNum-1 DO
	fbAlarmLogger[i](xEnable:=TRUE);
END_FOR
FOR i:=0 TO uiMessageEventNum-1 DO
	fbMessageLogger[i](xEnable:=TRUE);
END_FOR

METHOD M_ExportLoggedEvent_Off : BOOL
VAR_INPUT
END_VAR
fbExporter.xExecute			:= false;
END_METHOD

METHOD M_ExportLoggedEvent_On : BOOL
VAR_INPUT
	eEventExportType	:E_EventExportType;
	sFilePath			:STRING;
END_VAR
VAR_OUTPUT
	iResult:INT;
END_VAR
fbExporter.eEventExportType := eEventExportType;
fbExporter.sFilePath		:= sFilePath;

fbExporter.xExecute			:= TRUE;
END_METHOD

METHOD M_ExportLoggedEvent_State : BOOL
VAR_OUTPUT
	xBusy		:BOOL;
	xDone		:BOOL;
	xError		:BOOL;
END_VAR
xBusy	:= fbExporter.xBusy;
xDone	:= fbExporter.xDone;
xError	:= fbExporter.xError;
END_METHOD

METHOD M_AlarmEvent_Init : BOOL
VAR_INPUT
	fbDevice 	:REFERENCE TO FB_ActionBasic_Logger;
	Event		:TcEventEntry;
	uiIndex		:UINT;
END_VAR

(* Set Event *)
fbAlarmLogger[uiIndex].M_SetAlarmEvent(Event);


(* Connect to Device *)
fbDevice.M_ConnectAlarmLogger(fbAlarmLogger[uiIndex]);
END_METHOD

METHOD M_MessageEvent_Init : BOOL
VAR_INPUT
	fbDevice 	:REFERENCE TO FB_ActionBasic_Logger;
	Event		:TcEventEntry;
	uiIndex		:UINT;
END_VAR
(* Set Event *)
fbMessageLogger[uiIndex].M_SetMessageEvent(Event);


(* Connect to Device *)
fbDevice.M_ConnectMsgLogger(fbMessageLogger[uiIndex]);
END_METHOD

END_PROGRAM

// EventLogger/FB_EventLogger_Alarm
FUNCTION_BLOCK FB_EventLogger_Alarm EXTENDS FB_ActionBasic IMPLEMENTS ITF_EventLogger_Alarm
VAR_INPUT
	xEnable	:BOOL;
END_VAR
VAR_OUTPUT
END_VAR
VAR
	//State Machine
	StateBehaviour           : CBML.LConC;
	
	
	//Fb
	fbTcAlarm			:FB_TcAlarm;
	fbTcSourceInfo		:FB_TcSourceInfo;
	
	//Parameter
	Event				:TcEventEntry;
	
	
	//hr 					:HRESULT;
END_VAR

(*-----CBML State Machine-----*)
THIS^.IBehaviourModel := StateBehaviour;
StateBehaviour(xEnable:= xEnable, xBusy=> xBusy, xError=> xError);

METHOD M_ClearAlarm : BOOL
VAR
	hr 					:HRESULT;
END_VAR
VAR_OUTPUT
    iErrorID : INT := 0;
END_VAR
hr:=fbTcAlarm.Clear(0,TRUE);
		
IF FAILED(hr) THEN
	iErrorID:=9100;
ELSE
	iErrorID:=0;
END_IF
END_METHOD

METHOD M_ConfirmAlarm : BOOL
VAR
	hr 					:HRESULT;
END_VAR
VAR_OUTPUT
    iErrorID : INT := 0;
END_VAR
hr := fbTcAlarm.Confirm(0);
		
IF FAILED(hr) THEN
	iErrorID:=9200;
ELSE
	iErrorID:=0;
END_IF
END_METHOD

METHOD M_RaiseAlarm : BOOL
VAR_INPUT
	sSource_Name	: STRING(255);
	nSource_Id		: UDINT;
	sLogMessage		: T_MaxString;
END_VAR
VAR_OUTPUT
    iErrorID 		: INT := 0;
END_VAR
VAR
	hr 				:HRESULT;
END_VAR
fbTcSourceInfo.Clear();
		
fbTcSourceInfo.sName	:=sSource_Name;
fbTcSourceInfo.nId		:=nSource_Id;

//Create
IF NOT fbTcAlarm.EqualsToEventEntryEx(Event) THEN
	hr := fbTcAlarm.CreateEx(Event,TRUE,fbTcSourceInfo);
END_IF

IF FAILED(hr) THEN
	iErrorID:=9300;
ELSE
	//Add String
	fbTcAlarm.ipArguments.Clear().AddString(sLogMessage);
	
	//Raise
	hr := fbTcAlarm.Raise(0);
	
	IF FAILED(hr) THEN
		iErrorID:=9310;
	ELSE
		iErrorID:=0;
	END_IF
END_IF
END_METHOD

METHOD M_SetAlarmEvent : BOOL
VAR_INPUT
	Event	: TcEventEntry;
END_VAR
VAR_OUTPUT
    iErrorID : INT;
END_VAR
THIS^.Event := Event;
iErrorID:=0;
END_METHOD

PROPERTY pAlarmState : ST_AlarmEvent_State
GET
VAR
	stAlarmEventState	:ST_AlarmEvent_State;
END_VAR
stAlarmEventState.bActive				:=THIS^.fbTcAlarm.bActive;           
stAlarmEventState.bRaised				:=THIS^.fbTcAlarm.bRaised;           
stAlarmEventState.eConfirmnState		:=THIS^.fbTcAlarm.eConfirmationState;
stAlarmEventState.nTimeCleared			:=THIS^.fbTcAlarm.nTimeCleared;      
stAlarmEventState.nTimeConfirm			:=THIS^.fbTcAlarm.nTimeConfirmed;    
stAlarmEventState.nTimeRaised			:=THIS^.fbTcAlarm.nTimeRaised;       

pAlarmState := stAlarmEventState;
END_GET
END_PROPERTY

END_FUNCTION_BLOCK

// EventLogger/FB_EventLogger_Message
FUNCTION_BLOCK FB_EventLogger_Message EXTENDS FB_ActionBasic IMPLEMENTS ITF_EventLogger_Message
VAR_INPUT
	xEnable	:BOOL;
END_VAR
VAR_OUTPUT
END_VAR
VAR
	//State Machine
	StateBehaviour           : CBML.LConC;
	
	//Fbs
	fbTcMessage			:FB_TcMessage;
	fbTcSourceInfo		:FB_TcSourceInfo;
	
	//Para
	Event				:TcEventEntry;
	
END_VAR

(*-----CBML State Machine-----*)
THIS^.IBehaviourModel := StateBehaviour;
StateBehaviour(xEnable:= xEnable, xBusy=> xBusy, xError=> xError);

METHOD M_AddEventMsg : BOOL
VAR_INPUT
	//Event			: TcEventEntry;
	sSource_Name	: STRING(255);
	nSource_Id		: UDINT;
	sLogMessage		:T_MaxString;
END_VAR
VAR_OUTPUT
	iErrorID : INT := 0;
END_VAR
VAR
	hr 		: HRESULT;
END_VAR
fbTcSourceInfo.Clear();
fbTcSourceInfo.sName	:=sSource_Name;
fbTcSourceInfo.nId		:=nSource_Id;

//Create
hr := fbTcMessage.CreateEx(Event,fbTcSourceInfo);

IF FAILED(hr) THEN
	iErrorID := 9001;
ELSE
	
	//Text Argument
	fbTcMessage.ipArguments.Clear().AddString(sLogMessage);
	
	//Send
	hr := fbTcMessage.Send(0);
	
	IF FAILED(hr) THEN
		iErrorID := 9002;
	END_IF
END_IF
END_METHOD

METHOD M_SetMessageEvent : BOOL
VAR_INPUT
	Event	: TcEventEntry;
END_VAR
VAR_OUTPUT
	iErrorID	: INT;
END_VAR
THIS^.Event := Event;
iErrorID:=0;
END_METHOD

END_FUNCTION_BLOCK

// EventLogger/FB_EventLogger_Exporter
FUNCTION_BLOCK FB_EventLogger_Exporter EXTENDS FB_ActionBasic
VAR_INPUT
	xExecute			:BOOL;
	sFilePath			:STRING;
	eEventExportType	:E_EventExportType;
END_VAR
VAR_OUTPUT
END_VAR
VAR
	//State Machine
	StateBehaviour           : CBML.ETrig;
	
	//FBs
	fbEventLogger		: FB_TcEventLogger;
	fbCsvExportSetting	: FB_TcEventCsvExportSettings; 
	fbExportFilter		: FB_TcEventFilter; 
	
	//Para
	//sFilePath_Set			:STRING;
	eLanguage_Set			:E_EventLanguage:=E_EventLanguage.English;
	//eEventExportType_Set	:E_EventExportType;
	
	//Step
	iExport_Step			:INT;
END_VAR

(*-----CBML State Machine-----*)
THIS^.IBehaviourModel := StateBehaviour;
StateBehaviour(xExecute:= xExecute, xDone=> xDone, xBusy=> xBusy, xError=> xError);

METHOD CleanupAction
VAR_INPUT
    xAbortProposed : BOOL;
    iErrorIDProposed: INT;
END_VAR
VAR_OUTPUT
    xComplete : BOOL := TRUE;
    xAbort: BOOL := xAbortProposed;
 	iErrorID : INT := iErrorIDProposed;
END_VAR
iExport_Step:=0;
END_METHOD

METHOD CyclicAction
VAR_INPUT
    itfTimingController : CBML.ITimingController;
END_VAR
VAR_OUTPUT
    xComplete : BOOL := TRUE;
    iErrorID : INT := 0;
END_VAR
VAR
	bError	:BOOL;
	hr		:HRESULT;
END_VAR
xComplete:=FALSE;

CASE iExport_Step OF
	10://Export Settings
	
		//Set Output Event Language
		M_SetExportLanguage(eLanguage:=eLanguage_Set);
		
		//Set Output type
		M_SetExportParameter(eEventExportType:=eEventExportType);
		
		//CSV Output Setting
		M_SetCSV();
		
		IF fbCsvExportSetting.AddFilter(fbExportFilter) = S_OK THEN
			iExport_Step:=20;
		ELSE
			iErrorID := 9910;
			iExport_Step:=99;
		END_IF
		
	20://Export File
	
		IF fbEventLogger.ExportLoggedEvents(sFileName:= sFilePath, ipExportSettings:= fbCsvExportSetting, bError=> bError, hrErrorCode=> hr) THEN
			
			IF NOT bError THEN
				iExport_Step:=30;
			ELSE
				iErrorID:=TO_INT(hr);
				iExport_Step:=99;
			END_IF
			
		END_IF
	30://Done
		xComplete:=TRUE;
	99://Error
		xComplete:=TRUE;
END_CASE
END_METHOD

METHOD StartAction
VAR_OUTPUT
    xComplete : BOOL := TRUE;
	iErrorID : INT := 0;
END_VAR
iExport_Step:=10;
END_METHOD

METHOD PRIVATE M_SetCSV : BOOL
VAR_INPUT
END_VAR
fbCsvExportSetting.bWithHeader:=TRUE;
//fbCsvExportSetting.nLangId:=1033;
//fbCsvExportSetting.sDelimiter:=';';
END_METHOD

METHOD PRIVATE M_SetExportLanguage : BOOL
VAR_INPUT
	eLanguage	:E_EventLanguage;
END_VAR
fbCsvExportSetting.Clear();

CASE eLanguage OF
	E_EventLanguage.Chinese:
		fbCsvExportSetting.AddLanguage(TcLcid.zh_Hant, 'Chinese');
	E_EventLanguage.English:
		fbCsvExportSetting.AddLanguage(TcLcid.en_US, 'English');
	E_EventLanguage.German:
		fbCsvExportSetting.AddLanguage(TcLcid.de_DE, 'German');
END_CASE
END_METHOD

METHOD PRIVATE M_SetExportParameter : BOOL
VAR_INPUT
	eEventExportType	:E_EventExportType;
END_VAR
fbExportFilter.Clear();

CASE eEventExportType OF
	E_EventExportType.Message_And_Alarm:
		fbExportFilter.IsMessage().OR_OP().IsAlarm();
	E_EventExportType.Alarm:
		fbExportFilter.IsAlarm();
	E_EventExportType.Message:
		fbExportFilter.IsMessage();
END_CASE
END_METHOD

END_FUNCTION_BLOCK

// POUs/Demo
PROGRAM Demo
VAR
	//fbOneTimeProcess : FB_OneTimeExecute;
	fbCylinder : FB_Cylinder;
	FrontSR :BOOL;
	RearSR:BOOL;
	ExtendValve : BOOL;
	RetractValve:BOOL;
	SetupCylinderPara : ST_CylinderPara;
	SetupMotorPara : ST_MotorPara;
	bReset_gb:BOOL;
	MotorCtrl : FB_Motor;
END_VAR

SetupCylinderPara.ExtendTime:= T#400MS;
SetupCylinderPara.RetractTime := T#400MS;
SetupCylinderPara.ExtendDelayTime:=T#2S;
SetupCylinderPara.RetractDelayTime:=T#2S;
SetupCylinderPara.ExtendOverTime := T#5S;
SetupCylinderPara.RetractOverTime:=T#5S;
fbCylinder(
	xDone=> , 
	xBusy=> , 
	xError=> , 
	xEnable:= , 
	FrontSensor:= , 
	RearSensor:= RearSR,
	SetupPara := SetupCylinderPara,
	CurrentCylinderType=> , 
	InFrontPosition=> , 
	InRearPosition=> , 
	ExtendOutput=> ExtendValve, 
	RetractOutput=> );
	
SetupMotorPara.AccelerationTime := T#1S;
SetupMotorPara.DecelerationTime := T#1S;
MotorCtrl(
	xDone=> , 
	xBusy=> , 
	xError=> , 
	xEnable:= , 
	OverLoadSignal:= , 
	SetupPara:= SetupMotorPara, 
	InForWard=> , 
	InBackWard=> , 
	ForWardOutput=> , 
	BackWardOutput=> );	
IF bReset_gb THEN
	fbCylinder.M_Reset();
	MotorCtrl.M_Reset();
END_IF

END_PROGRAM

// EventLogger/_Test/FB_LoggerTest
FUNCTION_BLOCK FB_LoggerTest EXTENDS FB_ActionBasic_Logger
VAR_INPUT
END_VAR
VAR_OUTPUT
END_VAR
VAR
END_VAR

END_FUNCTION_BLOCK

// JsonMsgLogger/_Interface/Client/ITF_GetJsonMsg_Behavior
INTERFACE ITF_GetJsonMsg_Behavior

METHOD M_GetJsonMsg : BOOL
VAR_OUTPUT
	stJsonMsg	: ST_Json_MsgLogger;
	uiResult	: UINT;
END_VAR
END_METHOD

END_INTERFACE

// JsonMsgLogger/_Interface/Server/ITF_JsonMsg_Handler
INTERFACE ITF_JsonMsg_Handler

METHOD M_AttachJsonMsgLogger : BOOL
VAR_INPUT
	IDevice		:ITF_JsonMsg_Logger;
END_VAR
END_METHOD

END_INTERFACE

// JsonMsgLogger/_Test/Demo_JsonMsg
PROGRAM Demo_JsonMsg
VAR
	fbUserFunc			:ARRAY[0..5] OF FB_UserUnit;
	fbUserFunc2			:ARRAY[0..5] OF FB_UserUnit;
END_VAR
VAR
	bInitialized		:BOOL;
	i					:UINT;
	bTest				:BOOL;
	fbTimer				:TON;
	udAddCount			:UDINT;
	uiResult			:UINT;
END_VAR

(* ----------- 1. Function Call -----------*)
PRG_JsonMsg();

IF NOT bInitialized THEN
	bInitialized:=TRUE;
	
	(* ----------- 2. Set FilePath -----------*)
	PRG_JsonMsg.M_JsonMsg_SetFilePath(0,'C:\TwinCAT\3.1\Boot','LogMessage');
	PRG_JsonMsg.M_JsonMsg_SetFilePath(1,'C:\TwinCAT\3.1\Boot','LogMessage222');
	
	(* ----------- 3. Connect to Logger and Attach Logger to Handler -----------*)
	PRG_JsonMsg.M_JsonMsg_Init(fbUserFunc[0],0,0);
	PRG_JsonMsg.M_JsonMsg_Init(fbUserFunc[1],0,1);
	PRG_JsonMsg.M_JsonMsg_Init(fbUserFunc[2],0,2);
	PRG_JsonMsg.M_JsonMsg_Init(fbUserFunc[3],0,3);
	
	PRG_JsonMsg.M_JsonMsg_Init(fbUserFunc2[0],1,4);
	PRG_JsonMsg.M_JsonMsg_Init(fbUserFunc2[1],1,5);
	PRG_JsonMsg.M_JsonMsg_Init(fbUserFunc2[2],1,6);
	PRG_JsonMsg.M_JsonMsg_Init(fbUserFunc2[3],1,7);

END_IF

fbTimer(IN:= TRUE, PT:= T#100MS, Q=> , ET=> );

IF bTest AND fbTimer.Q THEN
	
	fbTimer(IN:= FALSE);

	fbUserFunc[0].M_AddJsonMsg('Handler_0');
	fbUserFunc2[0].M_AddJsonMsg('Handler_1');
END_IF

END_PROGRAM

// JsonMsgLogger/PRG_JsonMsg
PROGRAM PRG_JsonMsg
VAR
	fbJsonMsgHandler		:ARRAY[0..uiHandlerNum-1] OF FB_JsonMsg_Handler;
	fbJsonMsgLogger			:ARRAY[0..uiLoggerNum-1] OF FB_JsonMsg_Logger;
	fbGetTime				:NT_GetTime;
END_VAR
VAR
	i		:UINT;
END_VAR


(* -------FB refresh-------*)
fbGetTime(START:=NOT fbGetTime.START);

(* Handler *)
FOR i:=0 TO uiHandlerNum - 1 DO
	fbJsonMsgHandler[i](xEnable:=TRUE);
END_FOR

(* Logger *)
FOR i:=0 TO uiLoggerNum - 1 DO
	fbJsonMsgLogger[i](xEnable:=TRUE,timeNow:=fbGetTime.TIMESTR);
END_FOR

METHOD M_JsonMsg_Init : BOOL
VAR_INPUT
	fbDevice 				:REFERENCE TO FB_ActionBasic_Logger;
	
	uiHandlerIndex			:UINT;
	uiLoggerIndex			:UINT;
END_VAR
(* ----------- Connect to Logger ----------- *)
fbDevice.M_ConnectJsonMsgLogger(fbJsonMsgLogger[uiLoggerIndex]);


(* ----------- Connect to Logger ----------- *)
fbJsonMsgHandler[uiHandlerIndex].M_AttachJsonMsgLogger(fbDevice.itfJsonMsgLogger);
END_METHOD

METHOD M_JsonMsg_SetFilePath : BOOL
VAR_INPUT
	uiHandlerIndex			:UINT;
	sHandlerFilePath		:STRING;
	sHandlerFileName		:STRING;
END_VAR
fbJsonMsgHandler[uiHandlerIndex].M_SetFilePath(sHandlerFilePath,sHandlerFileName);
END_METHOD

END_PROGRAM

// JsonMsgLogger/FB_JsonMsg_Handler
FUNCTION_BLOCK FB_JsonMsg_Handler EXTENDS FB_ActionBasic IMPLEMENTS ITF_JsonMsg_Handler
VAR_INPUT
	xEnable		:BOOL;
END_VAR
VAR_OUTPUT
END_VAR
VAR
	//State Machine
	StateBehaviour			: CBML.LConC;
	
	itfJsonMsgLogger		:ARRAY[0..uiLoggerInHandlerMaxNum-1] OF ITF_JsonMsg_Logger;
	
	(* -----FBs----- *)
	fbQueue					: FB_Queue;				//Queue
	fbMemRingBuffer			: FB_MemRingBuffer;		//MemRing
	fbJsonConverter			: FB_Json_Converter;
	
	//File
	fbGetTime			: NT_GetTime;
	fbFileOpenTimer		: TON;
	fbFileCloseTimer	: TON;
	fbFileOpen 			: FB_FileOpen;
	fbFileWrite 		: FB_FileWrite;
	fbFileClose 		: FB_FileClose;
	fbFileRead			: FB_FileRead;
	tTimeNow			: TIMESTRUCT;
	
	(* -----Parameter----- *)
	sFileFolder			:T_MaxString;
	sFileName			:T_MaxString:='MessageLog';
	tFileOpenTime		:TIME:=T#30S;
	tFileCloseTime		:TIME:=T#1S;
	
	byteBuffer				:ARRAY[1..uiHandlerRingBufferSize-1] OF BYTE;
	
	addMessage			:ST_Json_MsgLogger;
	getMessage			:ST_Json_MsgLogger;
	stMsgFromLogger		:ST_Json_MsgLogger;
	sFilePath			:T_MaxString;
	bFileExist			:BOOL;
	sJsonString_FromObj	: STRING(10000);
	
	//-----Var-----
	iStep				:INT;
	uWriteCountTmp		:UINT;
	uWriteCount			:UINT;
	
END_VAR
VAR
	i,k						:UINT;
	uiTempNum				:UINT:=0;
	uiLoggerIndexNow		:UINT:=0;
	uiValidInterfaceNum		:UINT:=0;
END_VAR

(*-----CBML State Machine-----*)
THIS^.IBehaviourModel := StateBehaviour;
StateBehaviour(xEnable:= xEnable, xBusy=> xBusy, xError=> xError);


(* -----Logged Message Handle----- *)
M_HandleMessage();


(*-----FB refresh-----*)
fbGetTime(START:= NOT fbGetTime.START,TIMESTR=>tTimeNow);
fbJsonConverter();
fbMemRingBuffer();

fbFileOpen();
fbFileRead();
fbFileWrite();
fbFileClose();

METHOD CleanupAction
VAR_INPUT
    xAbortProposed : BOOL;
    iErrorIDProposed: INT;
END_VAR
VAR_OUTPUT
    xComplete : BOOL := TRUE;
    xAbort: BOOL := xAbortProposed;
 	iErrorID : INT := iErrorIDProposed;
END_VAR
//if file is writing => Wait Write
IF NOT fbFileWrite.bBusy THEN
	
	//Close File
	fbFileClose(hFile:= fbFileOpen.hFile, bExecute:= TRUE);
			
	IF (NOT fbFileClose.bBusy AND NOT fbFileClose.bError)		//File Close Done
	OR (fbFileClose.bError AND fbFileClose.nErrId = 1795) THEN//File has already been closed
	
		fbFileClose.bExecute:=FALSE;
		xComplete:=TRUE;
		
	ELSE//Not Finish
		
		xComplete:=FALSE;
		
	END_IF
END_IF
END_METHOD

METHOD CyclicAction
VAR_INPUT
    itfTimingController : CBML.ITimingController;
END_VAR
VAR_OUTPUT
    xComplete : BOOL := TRUE;
    iErrorID : INT := 0;
END_VAR
CASE iStep OF
	0:
		
	(* ---------- Check Lock State ----------*)
	100:
	
		IF eHandlerQueueType = E_HandlerQueueType.Queue THEN
			
			IF fbQueue.udiGetQueuedAmount > 0 THEN
				iStep:=200;
			END_IF
			
		ELSIF eHandlerQueueType = E_HandlerQueueType.RingBuffer THEN
			
			IF fbMemRingBuffer.nCount > 0 THEN
				iStep:=200;
			END_IF
			
		END_IF
	
	(* ---------- Check File Exist ----------*)
	200:
		sFilePath:=M_GetFilePathByTime(sFileFolder:=THIS^.sFileFolder,sFileName:=THIS^.sFileName);
		
		//Reset FBs 
		fbFileOpen.bExecute := FALSE;
		fbFileRead.bExecute := FALSE;
		fbFileWrite.bExecute := FALSE;
		fbFileClose.bExecute := FALSE;
		
		iStep:=210;
	210:
		fbFileOpen(
			sPathName:= sFilePath,
			nMode:=FOPEN_MODEREAD,
			ePath:= , 
			bExecute:= TRUE);
			
		IF NOT fbFileOpen.bBusy THEN
			
			fbFileOpen.bExecute := FALSE;
			
			IF fbFileOpen.bError THEN
				bFileExist:=FALSE;//File Not Exist
				iStep:=300;
			ELSE
				IF NOT (fbFileOpen.hFile = 0) THEN
					bFileExist:=TRUE;//File Exist
					iStep:=220;
				END_IF
			END_IF

		END_IF
	220:
		fbFileClose(
			hFile:= fbFileOpen.hFile, 
			bExecute:= TRUE);
			
		IF NOT fbFileClose.bBusy AND NOT fbFileClose.bError THEN
			fbFileClose.bExecute:=FALSE;
			iStep:=300;
		END_IF
	(* ---------- Append Data ----------*)
	300:
		fbFileOpen(
			sPathName:= sFilePath,
			nMode:=FOPEN_MODEAPPEND OR FOPEN_MODEPLUS,
			ePath:= , 
			bExecute:= TRUE);
			
		IF NOT fbFileOpen.bBusy THEN
			fbFileOpen.bExecute := FALSE;
			
			IF fbFileOpen.bError THEN
				iErrorID:=9300;
				iStep := 9999;
			ELSE
				IF NOT (fbFileOpen.hFile = 0) THEN
					
					uWriteCountTmp:=0;
					iStep := 310;
				END_IF
			END_IF
		END_IF
	310:
	
		//DeQueue
		IF eHandlerQueueType = E_HandlerQueueType.Queue THEN
			
			fbQueue.dequeueElement(pbtDequeueElement:=ADR(getMessage),udiDequeueSize:=SIZEOF(getMessage));
			
		ELSIF eHandlerQueueType = E_HandlerQueueType.RingBuffer THEN
			
			fbMemRingBuffer.A_RemoveHead(pRead:= ADR(getMessage),
										cbRead:= SIZEOF(getMessage),
										pBuffer:= ADR(byteBuffer),
										cbBuffer:= SIZEOF(byteBuffer),
										bOk=> );

		END_IF
		
		//Convert to Json String
		sJsonString_FromObj := fbJsonConverter.ObjToJsonStr(nData:= SIZEOF(getMessage), pData:= ADR(getMessage));
		
		IF bFileExist THEN
			sJsonString_FromObj:=CONCAT(',$N',sJsonString_FromObj);
		END_IF
		
		iStep := 320;
	
	320:
	
		fbFileWrite(
			hFile:= fbFileOpen.hFile, 
			pWriteBuff:= ADR(sJsonString_FromObj), 
			cbWriteLen:= LEN2(ADR(sJsonString_FromObj)), 
			bExecute:= TRUE);
		IF fbFileWrite.bError THEN
			fbFileWrite.bExecute:=FALSE;
			iErrorID:=9320;
			iStep := 9999;
		ELSIF NOT fbFileWrite.bBusy THEN
			bFileExist:=TRUE;
			fbFileWrite.bExecute:=FALSE;
			iStep := 330;
			uWriteCount:=uWriteCount+1;
		END_IF
	
	330:(* === Transition Condition ===*)
	
		//open file and write until 60s
		fbFileOpenTimer.IN:=TRUE;
		IF NOT fbFileOpenTimer.Q THEN
			
			IF eHandlerQueueType = E_HandlerQueueType.Queue THEN
			
				IF fbQueue.udiGetQueuedAmount > 0 THEN
					iStep:=310;				
				END_IF
				
			ELSIF eHandlerQueueType = E_HandlerQueueType.RingBuffer THEN
				
				IF fbMemRingBuffer.nCount > 0 THEN
					iStep:=310;				
				END_IF
			
			END_IF
		
		ELSE
			fbFileOpenTimer.IN:=FALSE;
			iStep:=340;
		END_IF
	
	(* ---------- Close File ----------*)
	340:
		fbFileClose(
			hFile:= fbFileOpen.hFile, 
			bExecute:= TRUE);
		IF fbFileClose.bError THEN
			iErrorID:=9340;
			iStep := 9999;
		ELSE
			iStep := 350;
		END_IF
	350:
		//close file for _s
		fbFileCloseTimer.IN:=TRUE;
		IF fbFileCloseTimer.Q THEN
			fbFileCloseTimer.IN:=FALSE;
			iStep:=100;
		END_IF
	(* ---------- State ----------*)
	9999://Error
		
END_CASE

fbFileCloseTimer(PT:= tFileCloseTime);
fbFileOpenTimer(PT:= tFileOpenTime);
END_METHOD

METHOD StartAction
VAR_OUTPUT
    xComplete : BOOL := TRUE;
	iErrorID : INT := 0;
END_VAR
iStep:=100;
END_METHOD

METHOD PRIVATE M_AddJsonMsg : BOOL
VAR_INPUT
	sLogMsg			:ST_Json_MsgLogger;
END_VAR
VAR_OUTPUT
	uiResult:UINT;
END_VAR
VAR
	hr	:UINT;
	bOk	:BOOL;
END_VAR
IF NOT xEnable THEN
	uiResult := 9001;
ELSE
	addMessage:=sLogMsg;
	
	
	IF eHandlerQueueType = E_HandlerQueueType.Queue THEN
		
		fbQueue.enqueueElement(iDataType:= 0, pbtEnqueue:=ADR(addMessage), udiEnqueueSize:= SIZEOF(addMessage),uiErrorID=>hr);
		
		IF hr = 0 THEN
			uiResult:=0;
		ELSE//Error
			IF hr = 771 THEN//Input = 0
				uiResult:=9771;
			ELSIF hr = 772 THEN//Size = 0
				uiResult:=9771;
			ELSIF hr = 773 THEN//non-matched data size
				uiResult:=9771;
			ELSE//Unknown
				uiResult:=9777;
			END_IF
		END_IF
		
	ELSIF eHandlerQueueType = E_HandlerQueueType.RingBuffer THEN
		
		fbMemRingBuffer.A_AddTail(pBuffer := ADR(byteBuffer), cbBuffer := SIZEOF(byteBuffer),pWrite := ADR(addMessage), cbWrite := SIZEOF(addMessage),bOk=> bOk,);
		
		IF bOk THEN
			uiResult:=0;(* Success *)
		ELSE
			uiResult:=9001;(* Buffer overflow *)
		END_IF
	END_IF
		
END_IF
END_METHOD

METHOD PRIVATE M_GetFilePathByTime : T_MaxString
VAR_INPUT
	sFileFolder	:T_MaxString;
	sFileName	:T_MaxString;
END_VAR
VAR
	sYear:STRING;
	sMon:STRING;
	sDay:STRING;
	sCombined:T_MaxString;
END_VAR

sYear:=TO_STRING(tTimeNow.wYear);
sMon:=TO_STRING(tTimeNow.wMonth);
sDay:=TO_STRING(tTimeNow.wDay);

sCombined:=CONCAT(sFileFolder,'\');
sCombined:=CONCAT(sCombined,sFileName);
sCombined:=CONCAT(sCombined,'_');


sCombined:=CONCAT(sCombined,sYear);

IF LEN(sMon) < 2 THEN
	sMon:=CONCAT('0',sMon);
END_IF
sCombined:=CONCAT(sCombined,sMon);

IF LEN(sDay) < 2 THEN
	sMon:=CONCAT('0',sDay);
END_IF
sCombined:=CONCAT(sCombined,sDay);


sCombined:=CONCAT(sCombined,'.json');
M_GetFilePathByTime:=sCombined;
END_METHOD

METHOD PRIVATE M_HandleMessage : BOOL
VAR_INPUT
END_VAR
(* -----Calc Valid Iterface num----- *)
uiTempNum:=0;
FOR i:=0 TO uiLoggerInHandlerMaxNum - 1 DO
	IF itfJsonMsgLogger[i] <> 0 THEN
		uiTempNum := uiTempNum + 1;
	ELSE
		EXIT;
	END_IF
END_FOR
IF uiValidInterfaceNum <> uiTempNum THEN
	uiValidInterfaceNum := uiTempNum;
END_IF

(* -----Message Handle----- *)
//one cycle deal with M Logger
FOR i := 0 TO uiLoggerHandleLimitPerCycle - 1 DO
	
	IF itfJsonMsgLogger[uiLoggerIndexNow] <> 0 THEN
		
		//Handler take N Msg from Logger one time
		FOR k:=0 TO uiMsgHandleLimitPerLogger - 1 DO
			
			IF itfJsonMsgLogger[uiLoggerIndexNow].pQueueAmount > 0 THEN//Data Exist in Logger
				
				IF eHandlerQueueType = E_HandlerQueueType.Queue THEN
					
					//Dequeue From Logger
					itfJsonMsgLogger[uiLoggerIndexNow].M_GetJsonMsg(stJsonMsg => stMsgFromLogger);
					
					//Enqueue to Master's Queue
					M_AddJsonMsg(stMsgFromLogger);
					
				ELSIF eHandlerQueueType = E_HandlerQueueType.RingBuffer THEN
					
					(* Check Volume *)
					IF fbMemRingBuffer.cbSize < (TO_LREAL(uiHandlerRingBufferSize) * 0.9) THEN
						
						//Dequeue From Logger
						itfJsonMsgLogger[uiLoggerIndexNow].M_GetJsonMsg(stJsonMsg => stMsgFromLogger);
						
						//Enqueue to Master's Queue
						M_AddJsonMsg(stMsgFromLogger);
						
					END_IF
				END_IF
			ELSE//Done
				EXIT;
			END_IF
			
		END_FOR
			
		//Calc Subject Index
		IF uiLoggerIndexNow < uiValidInterfaceNum - 1 THEN
			uiLoggerIndexNow := uiLoggerIndexNow + 1;
		ELSE
			uiLoggerIndexNow := 0;
		END_IF
	END_IF
	
END_FOR
END_METHOD

METHOD FB_init : BOOL
VAR_INPUT
	bInitRetains : BOOL; // if TRUE, the retain variables are initialized (warm start / cold start)
	bInCopyCode : BOOL;  // if TRUE, the instance afterwards gets moved into the copy code (online change)
END_VAR
IF eOsType = E_OS_Type.WinCE THEN
	THIS^.sFileFolder:= '\Hard Disk\TwinCAT\3.1\Boot';
ELSIF eOsType = E_OS_Type.Windows THEN
	THIS^.sFileFolder := 'C:\TwinCAT\3.1\Boot';
END_IF
END_METHOD

METHOD M_AttachJsonMsgLogger : BOOL
VAR_INPUT
	IDevice		:ITF_JsonMsg_Logger;
END_VAR
VAR
	i		:UINT;
END_VAR
FOR i:=0 TO uiLoggerInHandlerMaxNum - 1 DO
	IF IDevice <> 0 AND itfJsonMsgLogger[i] = 0 THEN
		itfJsonMsgLogger[i]:=IDevice;
		RETURN;
	END_IF
END_FOR
END_METHOD

METHOD M_SetFilePath : BOOL
VAR_INPUT
	sFileFolder	: Tc2_System.T_MaxString;
	sFileName	: Tc2_System.T_MaxString;
END_VAR
VAR_OUTPUT
	uiErrorCode	: UINT;
END_VAR
THIS^.sFileFolder	:= sFileFolder;
THIS^.sFileName		:= sFileName;
END_METHOD

END_FUNCTION_BLOCK

// JsonMsgLogger/Basic_Queue/FB_Queue
{attribute 'enable_dynamic_creation'}
//{attribute 'hide_all_locals'}
FUNCTION_BLOCK FB_Queue
VAR
	udiCount			:UDINT;
	bLinkList_Created	:BOOL;
	pHead				:POINTER TO ST_Queue;
	pTail				:POINTER TO ST_Queue;
	pReadCurrent		:POINTER TO ST_Queue;//leatest data pointer has been read
END_VAR

(*
Ver. 		: 1.2
Date 		: 2022/01/13
Content		: 
Ver1.2 Add error code for MEMCPY error
Ver1.1 edited changeCurrentbyIndex method line24
*)

METHOD dequeueElement : BOOL
VAR_INPUT
	pbtDequeueElement		: POINTER TO BYTE;//Pointer to Data e.g. ADR(Var)
	udiDequeueSize   		: UDINT;//Dequeued Data Size. e.g. sizeof(Var)
END_VAR
VAR_OUTPUT
	uiErrorID				: UINT;
END_VAR

VAR
	pTemp					: POINTER TO ST_Queue;
	udi2cpy					: UDINT;	
END_VAR
IF NOT checkInputErr(pbtInput:= pbtDequeueElement, udiSize:= udiDequeueSize, uiErrorID=> uiErrorID)THEN	
	RETURN;	
END_IF

IF udiCount<1 THEN
	uiErrorID:=768;//Link list not existed
	RETURN;
ELSIF udiCount=1 THEN
	pTemp:=pHead;
	pHead:=0;
	pTail:=0;
ELSIF udiCount>1 THEN
	pTemp:=pHead;		
	pHead:=pTemp^.pNext;
	pHead^.pPrev:=0;	
END_IF

IF pReadCurrent=pTemp THEN
	moveCurrent2Next(pReadCurrent); 
END_IF

udi2cpy:=MEMCPY(destAddr := pbtDequeueElement, srcAddr := pTemp^.pData, n := udiDequeueSize);
deleteElement(pTemp^.pData);
deleteElement(pTemp);
udiCount:=udiCount-1;
IF udiCount=0 THEN
	pReadCurrent:=0;
	bLinkList_Created:=FALSE;
END_IF

IF udi2cpy<>udiDequeueSize THEN
	uiErrorID:=773;//non-matched data size
END_IF

dequeueElement:=TRUE;
END_METHOD

METHOD enqueueElement : BOOL
VAR_INPUT
	iDataType		 : INT;//DataType Enum (user defined)
	pbtEnqueue 		 : POINTER TO BYTE;//Pointer to Data e.g. ADR(Var)
	udiEnqueueSize   : UDINT;//Enqueued Data Size. e.g. sizeof(Var)	
END_VAR
VAR_OUTPUT
	uiErrorID		 : UINT;
END_VAR
VAR
	pCurrent		 : POINTER TO ST_Queue;
	nCount			 : UDINT;
	udi2cpy			 : UDINT;	
END_VAR
IF NOT checkInputErr(pbtInput:= pbtEnqueue, udiSize:= udiEnqueueSize, uiErrorID=> uiErrorID)THEN	
	RETURN;
END_IF
 
IF udiCount=0 THEN
	pCurrent:=__NEW(ST_Queue);
	pHead:=pCurrent;
	pTail:=pCurrent;
	bLinkList_Created:=TRUE;
ELSIF udiCount>0 THEN
	pTail^.pNext:=__NEW(ST_Queue);
	pCurrent:=pTail^.pNext;
	pCurrent^.pPrev:=pTail;
	pTail:=pCurrent;
END_IF

pCurrent^.iDataType:=iDataType;
pCurrent^.pData:=__NEW(BYTE,udiEnqueueSize);
udi2cpy:=MEMCPY(destAddr := pCurrent^.pData, srcAddr := pbtEnqueue, n := udiEnqueueSize);
udiCount:=udiCount+1;

IF udi2cpy<>udiEnqueueSize THEN
	uiErrorID:=773;//non-matched data size
END_IF
enqueueElement:=true;
END_METHOD

METHOD enqueueElementfromHead : BOOL
VAR_INPUT
	iDataType			:INT;//DataType Enum (user defined)
	pbtEnqueue 			:POINTER TO BYTE;//Pointer to Data e.g. ADR(Var)
	udiEnqueueSize   	:UDINT;//Enqueued Data Size. e.g. sizeof(Var)
END_VAR
VAR_OUTPUT
	uiErrorID		 	: UINT;
END_VAR
VAR
	pCurrent			: POINTER TO ST_Queue;
	nCount				: UDINT;
	udi2cpy				: UDINT;	
	pOriginHead			: POINTER TO ST_Queue;
	pOriginTail			: POINTER TO ST_Queue;
END_VAR
IF NOT checkInputErr(pbtInput:= pbtEnqueue, udiSize:= udiEnqueueSize, uiErrorID=> uiErrorID)THEN	
	RETURN;
ELSE
	pOriginHead	:=pHead;
	pOriginTail	:=pTail;
END_IF

IF udiCount=0 THEN
	pCurrent:=__NEW(ST_Queue);
	pHead:=pCurrent;
	pTail:=pCurrent;
	bLinkList_Created:=TRUE;
ELSIF udiCount>0 THEN
	pHead^.pPrev:=__NEW(ST_Queue);
	pCurrent:=pHead^.pPrev;
	pCurrent^.pNext:=pHead;
	pHead:=pCurrent;
END_IF

pCurrent^.iDataType:=iDataType;
pCurrent^.pData:=__NEW(BYTE,udiEnqueueSize);
udi2cpy:=MEMCPY(destAddr := pCurrent^.pData, srcAddr := pbtEnqueue, n := udiEnqueueSize);
udiCount:=udiCount+1;

IF udi2cpy<>udiEnqueueSize THEN
	uiErrorID:=773;//non-matched data size
END_IF

enqueueElementfromHead:=TRUE;
END_METHOD

METHOD PUBLIC readElementbyIndex : BOOL
VAR_INPUT
	udiIndex					: UDINT;
	pbtReadElement			: POINTER TO BYTE;//Pointer to Data e.g. ADR(Var)
	udiReadSize   			: UDINT;//Read Data Size. e.g. sizeof(Var)
END_VAR
VAR_OUTPUT
	uiErrorID					: UINT;
END_VAR
VAR
	udi2cpy						: UDINT;
END_VAR
IF NOT checkInputErr(pbtInput:= pbtReadElement, udiSize:= udiReadSize, uiErrorID=> uiErrorID)THEN	
	RETURN;
END_IF

IF changeCurrentbyIndex(pChange:=pReadCurrent,udiIndex:= udiIndex,uiErrorID=>uiErrorID) THEN
	udi2cpy:=MEMCPY(destAddr := pbtReadElement, srcAddr := pReadCurrent^.pData, n := udiReadSize);
	IF udi2cpy<>udiReadSize THEN
		uiErrorID:=773;//non-matched data size
	END_IF
	readElementbyIndex:=TRUE;
END_IF
END_METHOD

METHOD PUBLIC readNextElement : BOOL
VAR_INPUT
	pbtReadElement				: POINTER TO BYTE;//Pointer to Data e.g. ADR(Var)
	udiReadSize   				: UDINT;//Read Data Size. e.g. sizeof(Var)
END_VAR
VAR_OUTPUT
	uiErrorID					: UINT;
END_VAR
VAR
	udi2cpy						: UDINT;
END_VAR
IF NOT checkInputErr(pbtInput:= pbtReadElement, udiSize:= udiReadSize, uiErrorID=> uiErrorID)THEN	
	RETURN;
END_IF

IF udiCount=0 THEN
	uiErrorID:=768;//Link list not existed
	pReadCurrent:=0;
	RETURN;
ELSIF pReadCurrent=0 THEN
	pReadCurrent:=pHead;
ELSE
	moveCurrent2Next(pReadCurrent);
END_IF


udi2cpy:=MEMCPY(destAddr := pbtReadElement, srcAddr := pReadCurrent^.pData, n := udiReadSize);
readNextElement:=TRUE;
IF udi2cpy<>udiReadSize THEN
	uiErrorID:=773;//non-matched data size
END_IF
END_METHOD

METHOD releaseQueue : BOOL
VAR
	pTemp				:POINTER TO ST_Queue;
	i					:UDINT;
END_VAR
VAR_OUTPUT
	uiErrorID			:UINT;
END_VAR
IF NOT bLinkList_Created THEN
	uiErrorID:=768;//Link list not existed
	RETURN;
END_IF

IF udiCount>1 THEN
	FOR i:= 1 TO udiCount-1 DO
		pTemp:=pHead;		
		pHead:=pTemp^.pNext;
		pHead^.pPrev:=0;	
		deleteElement(pTemp^.pData);
		deleteElement(pTemp);		
	END_FOR
END_IF	


//last data
pTemp:=pHead;
pHead:=0;
pTail:=0;
deleteElement(pTemp^.pData);
deleteElement(pTemp);
pReadCurrent:=0;
udiCount:=0;
bLinkList_Created:=FALSE;
releaseQueue:=TRUE;
END_METHOD

METHOD PRIVATE changeCurrentbyIndex : BOOL
VAR_INPUT
	udiIndex:UDINT;
END_VAR
VAR_IN_OUT
	pChange:POINTER TO ST_Queue;
END_VAR
VAR_OUTPUT
	uiErrorID:UINT;
END_VAR
VAR
	i:UDINT;
END_VAR
//2021.10.15 modify line 24 error (udiCount-udiIndex)

IF  udiCount=0  THEN
	uiErrorID:=768;//Link list not existed
	changeCurrentbyIndex:=FALSE;
	RETURN;
ELSIF udiIndex>udiCount OR udiIndex<1 THEN
	uiErrorID:=769;//Index not existed in list
	changeCurrentbyIndex:=FALSE;
	RETURN;
END_IF

IF udiIndex=1 THEN
	pChange:=pHead;
ELSIF udiIndex=udiCount THEN
	pChange:=pTail;
ELSIF (udiIndex-1)>=(udiCount-udiIndex) THEN
	pChange:=pHead;
	FOR i:=1 TO (udiIndex-1) DO
		moveCurrent2Next(pChange);
	END_FOR
ELSE
	pChange:=pTail;
	FOR i:=1 TO (udiCount-udiIndex) DO
		moveCurrent2Prev(pChange);
	END_FOR
END_IF
changeCurrentbyIndex:=true;
END_METHOD

METHOD PRIVATE checkInputErr : BOOL
VAR_INPUT
	pbtInput 	: POINTER TO BYTE;//Pointer to Data e.g. ADR(Var)
	udiSize   	: UDINT;//Enqueued Data Size. e.g. sizeof(Var)
END_VAR
VAR_OUTPUT
	uiErrorID	: UINT;
END_VAR
IF pbtInput=0 THEN
	uiErrorID:=771;
	RETURN;
ELSIF udiSize=0 THEN
	uiErrorID:=772;
	RETURN;
END_IF

checkInputErr:=TRUE;
END_METHOD

METHOD PRIVATE deleteElement : BOOL
VAR_INPUT
	pDelete		:POINTER TO ST_Queue;
END_VAR
VAR_OUTPUT
	uiErrorID:UINT;
END_VAR
IF pDelete<>0 THEN
	__DELETE(pDelete);
	pDelete:=0;
	deleteElement:=TRUE;
ELSE
	uiErrorID:=770;//Element already removed or not existed
END_IF
END_METHOD

METHOD PRIVATE moveCurrent2Next : BOOL
VAR_IN_OUT
	pMove:POINTER TO ST_Queue;
END_VAR
VAR_OUTPUT
	uiErrorID:UINT;
END_VAR
IF udiCount=0 THEN
	uiErrorID:=768;//Link list not existed
	pMove:=0;
	RETURN;
ELSIF pMove=pTail THEN
	pMove:=pHead;
ELSIF udiCount>0 AND pMove<>pTail THEN
	pMove:=pMove^.pNext;
END_IF
moveCurrent2Next:=TRUE;
END_METHOD

METHOD PRIVATE moveCurrent2Prev : BOOL
VAR_IN_out
	pMove:POINTER TO ST_Queue;
END_VAR
VAR_OUTPUT
	uiErrorID:UINT;
END_VAR
IF udiCount=0 THEN
	uiErrorID:=768;//Link list not existed
	pMove:=0;
	RETURN;
ELSIF pMove=pHead THEN
	pMove:=pTail;
ELSIF udiCount>=1 AND pMove<>pHead THEN
	pMove:=pMove^.pPrev;
END_IF
moveCurrent2Prev:=TRUE;
END_METHOD

PROPERTY PUBLIC bIsQueueCreated : bool
GET
bIsQueueCreated:=bLinkList_Created;
END_GET
SET
END_SET
END_PROPERTY

METHOD PUBLIC getDataTypebyIndex : BOOL
VAR_INPUT
	udiIndex:UDINT;
END_VAR
VAR_OUTPUT
	iDataType:INT;
	uiErrorID:UINT;
END_VAR
VAR
	pRead:POINTER TO ST_QUEUE;
END_VAR
IF changeCurrentbyIndex(pChange:=pRead,udiIndex:= udiIndex,uiErrorID=>uiErrorID) THEN
	iDataType:=pRead^.iDataType;
	getDataTypebyIndex:=TRUE;
END_IF
END_METHOD

METHOD PUBLIC getNextDataType : bool
VAR_OUTPUT
	iNextDataType:INT;
	uiErrorID:UINT;
END_VAR
IF pReadCurrent=0 AND udiCount=0 THEN
	uiErrorID:=768;//Link list not existed
	RETURN;
ELSIF pReadCurrent=0 AND udiCount<>0 THEN
	iNextDataType:=pHead^.iDataType;
	getNextDataType:=TRUE;
ELSIF pReadCurrent=pTail THEN
	iNextDataType:=pHead^.iDataType;
	getNextDataType:=TRUE;
ELSE
	iNextDataType:=pReadCurrent^.pNext^.iDataType;
	getNextDataType:=TRUE;
END_IF
END_METHOD

PROPERTY PUBLIC pGetHead : pointer to ST_QUEUE
GET
pGetHead:=pHead;
END_GET
SET
END_SET
END_PROPERTY

PROPERTY PUBLIC pGetTail : pointer to ST_QUEUE
GET
pGetTail:=pTail;
END_GET
SET
END_SET
END_PROPERTY

PROPERTY PUBLIC udiGetQueuedAmount : UDINT
GET
udiGetQueuedAmount:=udiCount;
END_GET
SET
END_SET
END_PROPERTY

END_FUNCTION_BLOCK

// JsonMsgLogger/Basic_Json/FB_Json_Converter
FUNCTION_BLOCK FB_Json_Converter
VAR_INPUT
END_VAR
VAR_OUTPUT
END_VAR
VAR
	// json功能块
	fbJsonRWDT 		: FB_JsonReadWriteDataType;
	fbJsonW 		: FB_JsonSaxPrettyWriter;
	fbJsonDP 		: FB_JsonDomParser;
END_VAR

(*
* 功能 1 输入键（字符串）-值（任意数据类型）自动载入json
* 功能 2 输入键（字符串）自动返回值（任意数据类型，包括自定义数据类型以及JSON）
* 功能 3 JSON数据重置
* 功能 4 输出JSON字符串
* 功能 5 输入JSON字符串，转化为Json对象（取消）
* 功能 6 输入特定结构体对象，直接转化为Json字符串并返回
* 功能 7 输入JSON字符串，转化为结构体
*)

METHOD JsonStrToObj : bool
VAR_INPUT
	JsonStr: STRING(10000);
	nData: UDINT;
	pData: PVOID;
END_VAR
VAR
	typestr: STRING;
	hrErrorCode : HRESULT;
END_VAR
(*
* 功能 7 输入JSON字符串，转化为结构体
*)
// 获得值变量的数据类型
typestr := fbJsonRWDT.GetDatatypeNameByAddress(nData := nData, pData := pData);
// 重置Json缓存
fbJsonW.ResetDocument();
// 将JSON字符串的信息写入特定数据
fbJsonRWDT.SetSymbolFromJson(sJson:= JsonStr, sDatatype:= typestr, nData:= nData, pData:= pData,hrErrorCode=>hrErrorCode);
END_METHOD

METHOD ObjToJsonStr : STRING(10000)
VAR_INPUT
	nData: UDINT;
	pData: PVOID;
END_VAR
VAR
	typestr: STRING;
END_VAR
(*
* 功能 6 输入特定结构体对象，直接转化为Json字符串并返回
*)
// 获得值变量的数据类型
typestr := fbJsonRWDT.GetDatatypeNameByAddress(nData := nData, pData := pData);
// 重置Json缓存
fbJsonW.ResetDocument();
//fbJsonW.SetFormatOptions(EJsonPrettyFormatOptions.eFormatSingleLineArray);
// 添加数据到Json缓存
fbJsonRWDT.AddJsonValueFromSymbol(fbJsonW, typestr, nData, pData);

// 将当前缓存转为字符串
fbJsonW.CopyDocument(pDoc:= ObjToJsonStr, nDoc:= SIZEOF(ObjToJsonStr));
END_METHOD

END_FUNCTION_BLOCK

// JsonMsgLogger/FB_JsonMsg_Logger
FUNCTION_BLOCK FB_JsonMsg_Logger EXTENDS FB_ActionBasic IMPLEMENTS ITF_JsonMsg_Logger
VAR_INPUT
	xEnable		:BOOL;
	timeNow		:TIMESTRUCT;
END_VAR
VAR_OUTPUT
END_VAR
VAR
	//State Machine
	StateBehaviour			: CBML.LConC;
	
	(* 3Ways(Loading Cost High to Low) *)
	fbQueue					: FB_Queue;												//Queue
	fbMemRingBuffer			: FB_MemRingBuffer;										//MemRing
	arrStoredJsonMsg		: ARRAY[0..uiBufferSize-1] OF ST_Json_MsgLogger;		//Fixed size Array
END_VAR
VAR
	(* Common Var *)
	count      				: UINT := 0; // now data Count
	addMessage				: ST_Json_MsgLogger;
	outMessage				: ST_Json_MsgLogger;
	
	(* MemRingBuffer Way *)
	byteBuffer				:ARRAY[1..uiRingBufferSize] OF BYTE;
	
	(* Fix Size way *)
	writeIndex 				: UINT := 0; // pos where Next data WRITE
    readIndex  				: UINT := 0; // pos where Next Data READ
    
END_VAR

(*-----CBML State Machine-----*)
THIS^.IBehaviourModel := StateBehaviour;
StateBehaviour(xEnable:= xEnable, xBusy=> xBusy, xError=> xError);

METHOD M_AddJsonMsg : BOOL
VAR_INPUT
	sLogMsg	: T_MaxString;
END_VAR
VAR_OUTPUT
	uiResult	: UINT;
END_VAR
VAR
	bOk	:BOOL;
END_VAR
CASE eLoggerQueueType OF
	E_LoggerQueueType.FixedSizeArray:
	
		IF count < uiBufferSize THEN
			arrStoredJsonMsg[writeIndex].sMessage	:= sLogMsg;
			arrStoredJsonMsg[writeIndex].tTime		:= SYSTEMTIME_TO_STRING(timeNow);
			writeIndex	:= (writeIndex + 1) MOD uiBufferSize;
			count := count + 1;
		(*
		//Overwrite Mode
		ELSIF count = uiBufferSize THEN
			
			readIndex := (readIndex + 1) MOD uiBufferSize;//Drop oldest data
			
			arrStoredJsonMsg[writeIndex].sMessage	:= sLogMsg;
			arrStoredJsonMsg[writeIndex].tTime		:= SYSTEMTIME_TO_STRING(fbGetTime.TIMESTR);
		
			writeIndex	:= (writeIndex + 1) MOD uiBufferSize;
		*)
		ELSE//Full
			uiResult:=9901;
		END_IF

	E_LoggerQueueType.Queue:
	
		addMessage.sMessage		:= sLogMsg;
		addMessage.tTime		:= SYSTEMTIME_TO_STRING(timeNow);
		fbQueue.enqueueElement(iDataType:=0,pbtEnqueue:=ADR(addMessage), udiEnqueueSize:= SIZEOF(addMessage),uiErrorID=>uiResult);
		count:=count+1;

	E_LoggerQueueType.RingBuffer:
	
		addMessage.sMessage		:= sLogMsg;
		addMessage.tTime		:= SYSTEMTIME_TO_STRING(timeNow);
		fbMemRingBuffer.A_AddTail(pBuffer := ADR(byteBuffer), cbBuffer := SIZEOF(byteBuffer),pWrite := ADR(addMessage), cbWrite := SIZEOF(addMessage),bOk=> bOk,);
		IF bOk THEN
			count:=count+1;
			uiResult:=0;(* Success *)
		ELSE
			uiResult:=9001;(* Buffer overflow *)
		END_IF
END_CASE
END_METHOD

METHOD M_GetJsonMsg : BOOL
VAR_OUTPUT
	stJsonMsg	: ST_Json_MsgLogger;
	uiResult	: UINT;
END_VAR
VAR
	bOk        : BOOL;
	uiErrorId	:UINT;
END_VAR
CASE eLoggerQueueType OF
	E_LoggerQueueType.FixedSizeArray:
	
		IF count > 0 THEN
			stJsonMsg := arrStoredJsonMsg[readIndex];
			readIndex := (readIndex + 1) MOD uiBufferSize;
			count := count - 1;
		ELSE//Empty
			uiResult:=9902;
		END_IF

	E_LoggerQueueType.Queue:
	
		fbQueue.dequeueElement(pbtDequeueElement:=ADR(stJsonMsg),udiDequeueSize:=SIZEOF(stJsonMsg),uiErrorID=>uiErrorId);
		
		IF uiErrorId <> 0 THEN
			uiResult:=0;
			count := count - 1;
		ELSE
			uiResult:=9902;
		END_IF
		

	E_LoggerQueueType.RingBuffer:
	
		fbMemRingBuffer.A_RemoveHead(pRead:= ADR(stJsonMsg),
						cbRead:= SIZEOF(stJsonMsg),
						pBuffer:= ADR(byteBuffer),
						cbBuffer:= SIZEOF(byteBuffer),
						bOk=> bOk);
								
		IF bOk THEN
			count := count - 1;
			uiResult:=0;(* Success *)
		ELSE
			uiResult:=9902;(* Buffer empty *)
		END_IF
END_CASE
END_METHOD

{warning 'add property implementation'}
PROPERTY pQueueAmount : UINT
GET
pQueueAmount:=count;
END_GET
END_PROPERTY

END_FUNCTION_BLOCK

// JsonMsgLogger/_Test/FB_UserUnit
FUNCTION_BLOCK FB_UserUnit EXTENDS FB_ActionBasic_Logger 
VAR_INPUT
END_VAR
VAR_OUTPUT
END_VAR
VAR
END_VAR

END_FUNCTION_BLOCK

// Utilities/FB_EdgeDetect
FUNCTION_BLOCK FB_EdgeDetect
VAR_INPUT
    xInput      : BOOL;     // 監視的布林輸入
END_VAR

VAR_OUTPUT
    xRisingEdge : BOOL;     // 上升沿輸出 (R_Trig)
    xFallingEdge: BOOL;     // 下降沿輸出 (F_Trig)
END_VAR

VAR
    xLastInput  : BOOL;     // 前一個週期的輸入狀態
END_VAR

// 程式邏輯
// 檢測上升沿 (FALSE -> TRUE)
xRisingEdge := xInput AND NOT xLastInput;

// 檢測下降沿 (TRUE -> FALSE)
xFallingEdge := NOT xInput AND xLastInput;

// 儲存當前輸入狀態供下一個週期使用
xLastInput := xInput;

END_FUNCTION_BLOCK
